(* Stoppen vom Prozess welches über den Automat ausgelöst wurde *)
	IF xTmpProcMachineStop THEN
		(* Step  function station stop  *)
		CASE iStepActionStop OF
		(* Überprüfe zuerst den Zustand des Prozesses ob es überhaupt zulässt, den Prozess zu stoppen *)
		1:	xTmp:=	TProcess.T_Ctrle.xRdy
					AND NOT(TProcess.T_Ctrle.xStop)
					AND NOT(TProcess.T_Ctrle.xDone)
					AND NOT(TProcess.T_Ctrle.xError)
					AND NOT(TProcess.T_Ctrle.xAbordProcess);
			IF xTmp THEN
				iStepActionStop:=10;
			(* not ready to execute stop *)
			ELSE iStepActionStop:=95; END_IF
		10:	TProcess.T_Ctrle.xStop:=TRUE;
			(* next step *)
			iStepActionStop:=20;
			xStepActionDoneStop:=FALSE;
		(* wait confirmation *)
		20:	T_ExchgParam.T_Visu.T_Message.iState:=232;	(* Warnung: Unverzüglicher Zyklus-Stopp ! *)
			IF NOT(xStepActionDoneStop) THEN
			(* release execution *)
				xStepActionDoneStop:=TRUE;
			ELSE
				IF NOT(TProcess.T_Ctrle.xStop) AND TProcess.T_Ctrle.xDone THEN
					(* Für Maschinenreferenzieren und Wstk Entlade Prozess wird der Prozess beendet *)
					xProcessAbordet:=TRUE;
					iStepActionStop:=90;
					xStepActionDoneStop:=FALSE;
					T_ExchgParam.T_Visu.T_Message.iState:=236;	(* Warnung: Prozess wurde gestoppt ! *)
				END_IF;
			END_IF;
		(* action done *)
		90:	xTmpProcMachineStop:=FALSE;
		(* function not ready *)
		95:	xTmpProcMachineStop:=FALSE;
		END_CASE;
	END_IF;
END_ACTION
ACTION VisuFunction_ProfileManagement:
(* Erstmalige Kopiervorgang der Profile *)
	IF xAction_CopyProfileToProcess THEN
		(* Set copy action *)
		CASE iStepAction OF
		(* Set default value *)
		1:	xFctSetDefaultValueStaticProfile(ptrT_DefaultProfileParameter:=ADR(T_Profile.T_DefaultProfileParameter));
			(* Init. display value *)
			xProfileFileNotFoundSt1:=FALSE;
			xWrongProfilNameReadedSt1:=FALSE;
			xProfileFileWrongSyntaxSt1:=FALSE;
			xProfileFileWrongSyntax:=FALSE;
			iStepAction:=2; (* Überprüfe zuerst als nächstes ob das USB Stick ansprechbar ist *)
		(* check first if USB-Stick exist *)
		2:	T_Profile.T_Ctrle.iFunction:=3;	(* check if the USB-Stick exist *)
			T_Profile.T_Ctrle.xExecute:=TRUE;
			iStepAction:=3;
		3:	IF NOT(T_Profile.T_Ctrle.xExecute) AND T_Profile.T_Ctrle.xDone THEN
				(* USB Stick exist *)
				iStepAction:=4;
			END_IF;
			IF NOT(T_Profile.T_Ctrle.xExecute) AND T_Profile.T_Ctrle.xErr THEN
				(* USB-Stick does not exist *)
				T_ExchgParam.T_Visu.T_Message.iState:=0;	(* Meldung zurücksetzen *)
				T_Profile.T_Ctrle.xReset:=TRUE;
				iStepAction:=98;
			END_IF;
		(* Read First all exist Profilname for manage the profile  *)
		4:	T_Profile.T_Ctrle.sPathAndFileName:='PROFILE\';
			T_Profile.T_Ctrle.iFunction:=6;
			T_Profile.T_Ctrle.xExecute:=TRUE;
			iStepAction:=5;
		5:	IF NOT(T_Profile.T_Ctrle.xExecute) AND T_Profile.T_Ctrle.xDone THEN
				(* all readed profile are ok *)
				iStepAction:=10;
			END_IF;
			IF NOT(T_Profile.T_Ctrle.xExecute) AND T_Profile.T_Ctrle.xErr THEN
				(* Wrong Syntax-->1 File of Profile is corrupted *)
				T_ExchgParam.T_Visu.T_Message.iState:=0;	(* Meldung zurücksetzen *)
				T_Profile.T_IDProfileStation[1].iNumber:=1;
				T_Profile.T_IDProfileStation[1].sName:='Default';
				T_Profile.T_Ctrle.xReset:=TRUE;
				xProfileFileWrongSyntax:=TRUE;
				iStepAction:=90;
			END_IF;
		(* activ reading profile file *)
		10:	IF T_NovRam.T_Parameter.T_StationWork[gciStationSt1].T_InfoProcess.iProfile > 0 AND T_NovRam.T_Parameter.T_StationWork[gciStationSt1].T_InfoProcess.iProfile <= csiMaxProfile THEN
				T_Profile.T_Ctrle.sPathAndFileName:='PROFILE\';
				T_Profile.T_Id.iNumber:=T_NovRam.T_Parameter.T_StationWork[gciStationSt1].T_InfoProcess.iProfile;
				T_Profile.T_Id.sName:=T_NovRam.T_Parameter.T_StationWork[gciStationSt1].T_InfoProcess.sProfileName;
				T_Profile.T_Ctrle.iFunction:=4;	(* read the profile file *)
				T_Profile.T_Ctrle.xExecute:=TRUE;
				(* next step *)
				iStepAction:=20;
			ELSE iStepAction:=25; END_IF
		20:	IF NOT T_Profile.T_Ctrle.xExecute AND T_Profile.T_Ctrle.xDone THEN
				(* Setzen des aktuellen Prozessabbild welches vom NovRAM ist *)
				T_Profile.T_LoadProfileParameter:=T_Profile.T_CopyProfileParameter;
				T_ExchgParam.T_StationCommon.T_Param_StationWork.T_InfoProcess.iProfile:=T_NovRam.T_Parameter.T_StationWork[gciStationSt1].T_InfoProcess.iProfile;
				T_ExchgParam.T_StationCommon.T_Param_StationWork.T_InfoProcess.sProfileName:=T_Profile.T_Id.sName;
				garPositionEndProcCalc[gciStationSt1]:=T_NovRam.T_Parameter.arZ1AxisCalcEndPosSaveProfile[gciStationSt1,T_NovRam.T_Parameter.T_StationWork[gciStationSt1].T_InfoProcess.iProfile];
				garCentringEndProcCalc[gciStationSt1]:=T_NovRam.T_Parameter.arZ1CentringCalcEndPosSaveProfile[gciStationSt1,T_NovRam.T_Parameter.T_StationWork[gciStationSt1].T_InfoProcess.iProfile];
				(* check if the read name of the profil file is the same as the save name *)
				IF (T_Profile.T_Ctrle.sProfileName <> T_Profile.T_Id.sName) THEN
					(* overwrite the profilname with the name wrote in the file *)
					T_NovRam.T_Parameter.T_StationWork[gciStationSt1].T_InfoProcess.sProfileName:=T_Profile.T_Ctrle.sProfileName;
					T_Profile.T_IDProfileStation[T_NovRam.T_Parameter.T_StationWork[gciStationSt1].T_InfoProcess.iProfile].sName:=T_Profile.T_Ctrle.sProfileName;
					xWrongProfilNameReadedSt1:=TRUE;
				END_IF;
				(* next step *)
				iStepAction:=90;
			END_IF
			IF T_Profile.T_Ctrle.xErr THEN
				iToLoadProfileNrSt1:=T_Profile.T_Id.iNumber;
				sToLoadProfileNameSt1:=T_Profile.T_Id.sName;
				IF (T_Profile.T_Ctrle.udiErrorID <> 16#F2000) THEN
					(* Profile file not founded *)
					xProfileFileNotFoundSt1:=TRUE;
				ELSE
					(* wrong syntax of readed Profile file *)
					xProfileFileWrongSyntaxSt1:=TRUE;
				END_IF;
				(* activ reset *)
				T_Profile.T_Ctrle.xReset:=TRUE;
				(* next step *)
				iStepAction:=25;
			END_IF
		(* waiting flag *)
		25:	IF NOT T_Profile.T_Ctrle.xReset AND T_Profile.T_Ctrle.xDone THEN
				IF (T_Profile.T_Id.iNumber = 1) THEN
					T_Profile.T_LoadProfileParameter:=T_Profile.T_DefaultProfileParameter;
					T_ExchgParam.T_StationCommon.T_Param_StationWork.T_InfoProcess.iProfile:=1;
					T_ExchgParam.T_StationCommon.T_Param_StationWork.T_InfoProcess.sProfileName:='Default';
					(* erase name *)
					T_Profile.T_IDProfileStation[1].sName:='Default';
					T_NovRam.T_Parameter.T_StationWork[gciStationSt1].T_InfoProcess.iProfile:=1;
					T_NovRam.T_Parameter.T_StationWork[gciStationSt1].T_InfoProcess.sProfileName:='Default';
					iStepAction:=90;
				ELSE
					(* erase name *)
					T_Profile.T_IDProfileStation[1].sName:='Default';
					T_NovRam.T_Parameter.T_StationWork[gciStationSt1].T_InfoProcess.iProfile:=1;
					T_NovRam.T_Parameter.T_StationWork[gciStationSt1].T_InfoProcess.sProfileName:='Default';
					iStepAction:=26;
				END_IF;
			END_IF
		(* activ reading profile file *)
		26:	T_Profile.T_Ctrle.sPathAndFileName:='PROFILE\';
			T_Profile.T_Id.iNumber:=1;
			T_Profile.T_Id.sName:='Default';
			T_Profile.T_Ctrle.iFunction:=4;	(* read the profile file *)
			T_Profile.T_Ctrle.xExecute:=TRUE;
			(* next step *)
			iStepAction:=20;
		(* End function *)
		90:	xTmp:=	xProfileFileNotFoundSt1 OR xWrongProfilNameReadedSt1 OR 	xProfileFileWrongSyntaxSt1 OR xProfileFileWrongSyntax;
			IF xTmp THEN
				IF xProfileFileNotFoundSt1 THEN
					T_ExchgParam.T_SafetyCtrl.diSetForceErrorNr:=(gciStationSt1 * 1000000) + 16#F301;	(* Datei für zu ladendes Profil nicht gefunden *)
				ELSE
					IF xWrongProfilNameReadedSt1 THEN
						T_ExchgParam.T_SafetyCtrl.diSetForceErrorNr:=(gciStationSt1 * 1000000) + 16#F303;	(* Profilname von Datei ist anders als geladenes Profil *)
					END_IF;
					IF xProfileFileWrongSyntaxSt1 THEN
						T_ExchgParam.T_SafetyCtrl.diSetForceErrorNr:=(gciStationSt1 * 1000000) + 16#F304;	(* Syntaxfehler von zu ladendes Profil *)
					END_IF;
					IF xProfileFileWrongSyntax THEN
						T_ExchgParam.T_SafetyCtrl.diSetForceErrorNr:=16#F303;	(* Syntaxfehler mindestens einer Profildatei beim lesen aller Profile *)
					END_IF;
				END_IF;
				T_ExchgParam.T_SafetyCtrl.xSetForceError:=TRUE;
				xProfileFileNotFoundSt1:=xWrongProfilNameReadedSt1:=xProfileFileWrongSyntaxSt1:=FALSE;
				xProfileFileWrongSyntax:=FALSE;
			END_IF;
			T_Visu.T_CtrleAction.xDone:=TRUE;
			T_Visu.T_CtrleAction.xErr:=FALSE;
			T_Visu.T_CtrleAction.udiErrorID:=16#0;
			xAction_CopyProfileToProcess:=FALSE;
			xUpdateProfileList:=TRUE;
		(* USB-Stick is missing  *)
		98:	T_Visu.T_CtrleAction.xDone:=TRUE;
			T_Visu.T_CtrleAction.xNotReady:=FALSE;
			T_Profile.T_Ctrle.xReset:=T_Profile.T_Ctrle.xErr;
			T_ExchgParam.T_SafetyCtrl.xSetForceError:=TRUE;
			T_ExchgParam.T_SafetyCtrl.diSetForceErrorNr:=16#F300;	(* USB-Stick konnte nicht gefunden werden für Profil lesen/schreiben *)
			T_Visu.T_CtrleAction.xErr:=FALSE;
			T_Visu.T_CtrleAction.udiErrorID:=0;
			xAction_CopyProfileToProcess:=FALSE;
		END_CASE
	END_IF

(* Laden eines ausgewählten Profil in den Prozessabbild *)
	IF xAction_LoadProfile THEN
		(* Step import/export profile value *)
		CASE iStepAction OF
		1:	IF NOT(T_NovRAM.T_Parameter.T_Machine.T_ParamSystem.xActive_ProfilLoadNormalMode) AND
			     NOT(gT_SafetyStatus.xSetupOperateModeActive) THEN
				T_ExchgParam.T_Visu.T_Message.iState:=250;	(* Warning: Laden Profile im Automat ist der Parameter gesperrt ! *)
				iStepAction:=90;
				RETURN;
			END_IF;
			T_ExchgParam.T_Visu.T_Message.iState:=104;	(* Aufforderung: Bestätigen Profil laden <Enter>, abbrechen <Esc> ? *)
			xWrongProfilNameReaded:=FALSE;
			xProfileFileNotFoundSt:=FALSE;
			xProfileFileWrongSyntax:=FALSE;
			(* next step *)
			iStepAction:=10;
		(* waiting for key <Enter> or <Esc> *)
		10:	IF RisingEdgeKeyPanel_Enter.Q THEN
				(* Display message transfering *)
				T_ExchgParam.T_Visu.T_Message.iState:=4;	(* Info: Übertragung von Werten... *)
				tTimeOutAction:=TimerAction.ET+T#10s;
				iStepAction:=11;
			ELSE
				IF RisingEdgeKeyPanel_Esc.Q THEN
					iStepAction:=90;
					T_ExchgParam.T_Visu.T_Message.iState:=202;	(* Warnung: Aktion abgebrochen ! *)
				END_IF
			END_IF
			(* An other message has been displayed *)
			IF (T_ExchgParam.T_Visu.T_Message.iState<>4) AND (T_ExchgParam.T_Visu.T_Message.iState<>104) AND (T_ExchgParam.T_Visu.T_Message.iState<>202) THEN iStepAction:=90; END_IF
		(* check first if USB-Stick exist *)
		11:	T_Profile.T_Ctrle.iFunction:=3;	(* check if the USB-Stick exist *)
			T_Profile.T_Ctrle.xExecute:=TRUE;
			iStepAction:=12;
		12:	IF NOT(T_Profile.T_Ctrle.xExecute) AND T_Profile.T_Ctrle.xDone THEN
				(* USB Stick exist *)
				IF (T_Profile.T_IDProfileStation[T_ExchgParam.T_ProfileCommon.T_Id.iNumber].sName = '') THEN
					T_ExchgParam.T_Visu.T_Message.iState:=218;		(* Warnung: Profil existiert nicht ! *)
					iStepAction:=90;
				ELSE
					iStepAction:=20;
				END_IF;
			END_IF;
			IF NOT(T_Profile.T_Ctrle.xExecute) AND T_Profile.T_Ctrle.xErr THEN
				(* USB-Stick does not exist *)
				T_ExchgParam.T_Visu.T_Message.iState:=0;	(* Meldung zurücksetzen *)
				T_Profile.T_Ctrle.xReset:=TRUE;
				iStepAction:=98;
			END_IF;
		(* Init. reading profile file *)
		20:	(* Save Old Slide Reference Position *)
			T_Profile.T_Ctrle.sPathAndFileName:='PROFILE\';
			T_Profile.T_Id.iNumber:=T_ExchgParam.T_ProfileCommon.T_Id.iNumber;
			T_Profile.T_Id.sName:=T_Profile.T_IDProfileStation[T_ExchgParam.T_ProfileCommon.T_Id.iNumber].sName;
			T_Profile.T_Ctrle.iFunction:=4;	(* read the profile file *)
			T_Profile.T_Ctrle.xExecute:=TRUE;
			(* Display info message *)
			T_ExchgParam.T_Visu.T_Message.iState:=4;	(* Info: Übertragung von Werten... *)
			(* next step *)
			iStepAction:=30;
		(* waiting confirmation signal *)
		30:	T_ExchgParam.T_Visu.T_Message.iState:=4;	(* Info: Übertragung von Werten... *)
			IF NOT T_Profile.T_Ctrle.xExecute AND T_Profile.T_Ctrle.xDone THEN
			(* Copy profile to online value *)
				T_NovRam.T_Parameter.T_StationWork[gciStationSt1].T_StProcess:=T_Profile.T_CopyProfileParameter.T_ProzessData;
				T_NovRam.T_Parameter.T_StationWork[gciStationSt1].T_OnlineChange:=T_Profile.T_CopyProfileParameter.T_ProfileOnlineChange;
				T_Profile.T_LoadProfileParameter:=T_Profile.T_CopyProfileParameter;
				IF (T_NovRam.T_Parameter.T_StationWork[gciStationSt1].T_InfoProcess.iProfile <> T_ExchgParam.T_ProfileCommon.T_Id.iNumber) THEN
					(* Anderes Profile geladen und deshalb muss der entsprechende Zählerstand des geladenen Profil übernommen werden *)
					garPositionEndProcCalc[gciStationSt1]:=T_NovRam.T_Parameter.arZ1AxisCalcEndPosSaveProfile[gciStationSt1,T_ExchgParam.T_ProfileCommon.T_Id.iNumber];
					garCentringEndProcCalc[gciStationSt1]:=T_NovRam.T_Parameter.arZ1CentringCalcEndPosSaveProfile[gciStationSt1,T_ExchgParam.T_ProfileCommon.T_Id.iNumber];
				END_IF;
				T_NovRam.T_Parameter.T_StationWork[gciStationSt1].T_InfoProcess.iProfile:=T_ExchgParam.T_ProfileCommon.T_Id.iNumber;
				T_NovRam.T_Parameter.T_StationWork[gciStationSt1].T_InfoProcess.sProfileName:=T_Profile.T_Id.sName;
				T_ExchgParam.T_ProfileCommon.T_OnlineChange.T_Data:=T_Profile.T_LoadProfileParameter.T_ProfileOnlineChange;
				T_ExchgParam.T_ProfileCommon.T_Id.sName:=T_Profile.T_Id.sName;
				T_ExchgParam.T_StationCommon.T_Param_StationWork.T_StProcess:=T_Profile.T_LoadProfileParameter.T_ProzessData;
				(* check if the read name of the profil file is the same as the save name *)
				IF (T_Profile.T_Ctrle.sProfileName <> T_Profile.T_Id.sName) THEN
					(* overwrite the profilname with the name wrote in the file *)
					T_NovRam.T_Parameter.T_StationWork[gciStationSt1].T_InfoProcess.sProfileName:=T_Profile.T_Ctrle.sProfileName;
					T_ExchgParam.T_ProfileCommon.T_Id.sName:=T_Profile.T_Ctrle.sProfileName;
					T_Profile.T_IDProfileStation[T_ExchgParam.T_ProfileCommon.T_Id.iNumber].sName:=T_Profile.T_Ctrle.sProfileName;
					xWrongProfilNameReaded:=TRUE;
				END_IF;
				(* next step *)
				iStepAction:=40;
			END_IF
			IF T_Profile.T_Ctrle.xErr THEN
				iToLoadProfileNrSt:=T_Profile.T_Id.iNumber;
				sToLoadProfileNameSt:=T_Profile.T_Id.sName;
				(* activ reset *)
				T_Profile.T_Ctrle.xReset:=TRUE;
				IF (T_Profile.T_Ctrle.udiErrorID <> 16#F2000) THEN
					(* Profile file not founded *)
					xProfileFileNotFoundSt:=TRUE;
					T_ExchgParam.T_ProfileCommon.T_Id.sName:='';
					(* Profile will be erased from the profile list *)
					T_Profile.T_IDProfileStation[T_ExchgParam.T_ProfileCommon.T_Id.iNumber].sName:='';
					xUpdateProfileList:=TRUE;
					(* next step *)
					iStepAction:=90;
				ELSE
					(* wrong syntax of readed Profile file *)
					xProfileFileWrongSyntax:=TRUE;
					(* next step *)
					iStepAction:=90;
				END_IF;
			END_IF
		(* save profile number *)
		40:	(* save profile number to process value *)
			T_ExchgParam.T_StationCommon.T_Param_StationWork.T_InfoProcess.iProfile:=T_ExchgParam.T_ProfileCommon.T_Id.iNumber;
			T_ExchgParam.T_StationCommon.T_Param_StationWork.T_InfoProcess.sProfileName:=T_ExchgParam.T_ProfileCommon.T_Id.sName;
			xUpdateHandlingConfig:=TRUE;
			(* activ next step *)
			iStepAction:=50;
		(* active saving data NovRAM *)
		50:	xAction_SaveNovRAM:=TRUE;
			xBlockSetNovRamAction_End:=TRUE;
			iStepActionNovRam:=1;
			(* next step *)
			iStepAction:=60;
		(* waiting confirm saving NovRAM action *)
		60:	IF NOT xAction_SaveNovRAM THEN
				T_ExchgParam.T_Visu.T_Message.iState:=54;	(* Info: Profil wurde geladen ! *)
				IF NOT(xProfileFileNotFoundSt) THEN
					iStepAction:=90;
				ELSE
					iStepAction:=90;
				END_IF;
			END_IF;
		(* save done *)
		90:	IF xProfileFileNotFoundSt OR xWrongProfilNameReaded OR xProfileFileWrongSyntax THEN
				IF xProfileFileNotFoundSt THEN
					T_ExchgParam.T_SafetyCtrl.diSetForceErrorNr:=(gciStationSt1 * 1000000) + 16#F301;	(* Datei für zu ladendes Profil nicht gefunden *)
				ELSE
					IF xWrongProfilNameReaded THEN
						T_ExchgParam.T_SafetyCtrl.diSetForceErrorNr:=(gciStationSt1 * 1000000) + 16#F303;	(* Profilname von Datei ist anders als geladenes Profil *)
					ELSE
						T_ExchgParam.T_SafetyCtrl.diSetForceErrorNr:=(gciStationSt1 * 1000000) + 16#F304;	(* Syntaxfehler von zu ladendes Profil *)
					END_IF;
				END_IF;
				T_ExchgParam.T_SafetyCtrl.xSetForceError:=TRUE;
				xProfileFileNotFoundSt:=xWrongProfilNameReaded:=xProfileFileWrongSyntax:=FALSE;
			END_IF;
			T_Visu.T_CtrleAction.xDone:=TRUE;
			T_Visu.T_CtrleAction.xNotReady:=FALSE;
			T_Visu.T_CtrleAction.xErr:=FALSE;
			T_Visu.T_CtrleAction.udiErrorID:=0;
			xAction_LoadProfile:=FALSE;
		(* USB-Stick is missing  *)
		98:	T_Visu.T_CtrleAction.xDone:=TRUE;
			T_Visu.T_CtrleAction.xNotReady:=FALSE;
			T_Profile.T_Ctrle.xReset:=T_Profile.T_Ctrle.xErr;
			T_ExchgParam.T_SafetyCtrl.xSetForceError:=TRUE;
			T_ExchgParam.T_SafetyCtrl.diSetForceErrorNr:=(gciStationSt1 * 1000000) + 16#F300;	(* USB-Stick konnte nicht gefunden werden für Profil lesen/schreiben *)
			T_Visu.T_CtrleAction.xErr:=FALSE;
			T_Visu.T_CtrleAction.udiErrorID:=0;
			xAction_LoadProfile:=FALSE;
		END_CASE
	ELSE
		IF NOT(xAction_CopyProfileToProcess) THEN
			IF (T_NovRam.T_Parameter.T_StationWork[1].T_InfoProcess.iProfile >= 1) AND (T_NovRam.T_Parameter.T_StationWork[1].T_InfoProcess.iProfile <= 100) THEN
				T_NovRam.T_Parameter.arZ1AxisCalcEndPosSaveProfile[gciStationSt1,T_NovRam.T_Parameter.T_StationWork[1].T_InfoProcess.iProfile]:=garPositionEndProcCalc[gciStationSt1];
				T_NovRam.T_Parameter.arZ1CentringCalcEndPosSaveProfile[gciStationSt1,T_NovRam.T_Parameter.T_StationWork[1].T_InfoProcess.iProfile]:=garCentringEndProcCalc[gciStationSt1];
			END_IF;
		END_IF;
	END_IF

(* Speichern eines ausgewählten Profils *)
	IF xAction_SaveProfile THEN
		(* Step saving NovRAM *)
		CASE iStepAction OF
		(* check first if USB-Stick exist *)
		1:	T_Profile.T_Ctrle.iFunction:=3;	(* check if the USB-Stick exist *)
			T_Profile.T_Ctrle.xExecute:=TRUE;
			iStepAction:=2;
		2:	IF NOT(T_Profile.T_Ctrle.xExecute) AND T_Profile.T_Ctrle.xDone THEN
				(* USB Stick exist *)
				iStepAction:=10;
			END_IF;
			IF NOT(T_Profile.T_Ctrle.xExecute) AND T_Profile.T_Ctrle.xErr THEN
				(* USB-Stick does not exist *)
				T_ExchgParam.T_Visu.T_Message.iState:=0;	(* Meldung zurücksetzen *)
				T_Profile.T_Ctrle.xReset:=TRUE;
				iStepAction:=98;
			END_IF;
		(* Display message to ask for confirmation *)
		10:	IF T_ExchgParam.T_ProfileCommon.T_Id.iNumber > 1 THEN
				IF T_ExchgParam.T_ProfileCommon.T_Id.sName <> '' THEN
					iTmp:=  iFctExistProfileName(	sProfileName:=T_ExchgParam.T_ProfileCommon.T_Id.sName,
												ptrProfileList:=ADR(T_Profile.T_IDProfileStation));
					IF iTmp = T_ExchgParam.T_ProfileCommon.T_Id.iNumber OR iTmp = 0 THEN
						IF (T_ExchgParam.T_StationCommon.T_Param_StationWork.T_InfoProcess.iProfile = T_ExchgParam.T_ProfileCommon.T_Id.iNumber) THEN
							(* Display message 'ask for rewriting' *)
							T_ExchgParam.T_Visu.T_Message.iState:=105;	(* Aufforderung: Das Profil wird überschrieben <Enter>, abbrechen <Esc> ? *)
							(* next step *)
							iStepAction:=20;
						ELSE
							(* Display message 'confirm saving' *)
							T_ExchgParam.T_Visu.T_Message.iState:=103;	(* Aufforderung: Speichern bestätigen <Enter>, abbrechen <Esc> ? *)
							(* next step *)
							iStepAction:=20;
						END_IF
					ELSE
						T_ExchgParam.T_Visu.T_Message.iState:=219;		(* Warnung: Profil existiert schon, Daten nicht gespeichert ! *)
						iStepAction:=90;
					END_IF;
				(* Display message, 'Profile name not correct' *)
				ELSE	T_ExchgParam.T_Visu.T_Message.iState:=220;		(* Warnung: Profilname nicht korrekt ! *)
						iStepAction:=90;
				END_IF
			ELSE
				T_ExchgParam.T_Visu.T_Message.iState:=221;	(* Warnung: Default-Profilwerte können nicht geändert werden ! *)
				iStepAction:=90;
			END_IF
		(* waiting for confirmation key <Enter> or <Esc> *)
		20:	IF RisingEdgeKeyPanel_Enter.Q THEN
			(* Display message *)
				T_ExchgParam.T_Visu.T_Message.iState:=3;		(* Info: Start speichern... *)
				tTimeOutAction:=TimerAction.ET+T#10s;
				(* next step *)
				iStepAction:=30;
			ELSE
				IF RisingEdgeKeyPanel_Esc.Q THEN
					iStepAction:=90;
					T_ExchgParam.T_Visu.T_Message.iState:=202;	(* Warnung: Aktion abgebrochen ! *)
				END_IF
			END_IF
			(* An other message has been displayed *)
			IF (T_ExchgParam.T_Visu.T_Message.iState<>3) AND (T_ExchgParam.T_Visu.T_Message.iState<>103) AND
			     (T_ExchgParam.T_Visu.T_Message.iState<>105) AND (T_ExchgParam.T_Visu.T_Message.iState<>202) THEN iStepAction:=90; END_IF
		30:	(* activ saving profile file *)
			T_Profile.T_Ctrle.sPathAndFileName:='PROFILE\';
			T_Profile.T_Id.iNumber:=T_ExchgParam.T_ProfileCommon.T_Id.iNumber;
			T_Profile.T_Id.sName:=T_ExchgParam.T_ProfileCommon.T_Id.sName;
			T_Profile.T_Ctrle.iFunction:=5;	(* write the profile file *)
			T_Profile.T_Ctrle.xExecute:=TRUE;
			T_Profile.T_CopyProfileParameter.T_ProzessData:=T_NovRam.T_Parameter.T_StationWork[gciStationSt1].T_StProcess;
			T_Profile.T_CopyProfileParameter.T_ProfileOnlineChange:=T_NovRam.T_Parameter.T_StationWork[gciStationSt1].T_OnlineChange;
			(* next step *)
			iStepAction:=40;
		(* waiting signal and start saving data in NovRAM *)
		40:	T_ExchgParam.T_Visu.T_Message.iState:=3;		(* Info: Start speichern... *)
			IF NOT(T_Profile.T_Ctrle.xExecute) AND T_Profile.T_Ctrle.xDone THEN
				T_Profile.T_IDProfileStation[T_ExchgParam.T_ProfileCommon.T_Id.iNumber]:=T_ExchgParam.T_ProfileCommon.T_Id;
				(* Process profile value = file profile value *)
				IF (T_ExchgParam.T_ProfileCommon.T_Id.iNumber = T_NovRam.T_Parameter.T_StationWork[gciStationSt1].T_InfoProcess.iProfile) THEN
					(* Beim speichern eines Profils darf dies nicht durchgeführt werden, sofern nicht das gleiche Profil gespeichert wird wo schon geladen ist,
					    weil sonst der Blaue Profilebalken überschrieben wird *)
					T_ExchgParam.T_StationCommon.T_Param_StationWork.T_InfoProcess.sProfileName:=T_ExchgParam.T_ProfileCommon.T_Id.sName;
					T_Profile.T_LoadProfileParameter:=T_Profile.T_ProcProfileParameter;
					T_NovRam.T_Parameter.T_StationWork[gciStationSt1].T_InfoProcess.sProfileName:=T_ExchgParam.T_ProfileCommon.T_Id.sName;
				END_IF
				(* page profile, update profile list *)
				xUpdateProfileList:=TRUE;
				(* next step *)
				iStepAction:=50;
			END_IF
			IF T_Profile.T_Ctrle.xErr THEN
				iStepAction:=98;
			END_IF
		(* save Image in NovRAM *)
		50:	T_NovRAM.T_Ctrle.xExecute:=TRUE;
			T_NovRAM.T_Ctrle.iFunction:=2;
			(* next Step *)
			iStepAction :=60;
			xStepActionDone:=FALSE;
		(* wait save confirmation *)
		60:	IF NOT(xStepActionDone) THEN
				T_NovRAM.T_Ctrle.xExecute:=FALSE;
				(* confirm Step *)
				xStepActionDone:=TRUE;
			ELSE
				IF T_NovRAM.T_Ctrle.xDone THEN
				(* next Step *)
					iStepAction :=90;
					xStepActionDone:=FALSE;
					T_ExchgParam.T_Visu.T_Message.iState:=55;	(* Info: Profil wurde gespeichert ! *)
				ELSE	IF T_NovRAM.T_Ctrle.xErr THEN
							iStepAction:=99;
							xStepActionDone:=FALSE;
						END_IF
				END_IF
			END_IF
		(* save done *)
		90:	T_Visu.T_CtrleAction.xDone:=TRUE;
			T_Visu.T_CtrleAction.xNotReady:=FALSE;
			T_Visu.T_CtrleAction.xErr:=FALSE;
			T_Visu.T_CtrleAction.udiErrorID:=0;
			xAction_SaveProfile:=FALSE;
		(* NovRAM not ready *)
		95:	TimerNotReady(IN:=TRUE);
			xAction_SaveProfile:=FALSE;
		(* USB-Stick is missing or directory is missing *)
		98:	T_Visu.T_CtrleAction.xDone:=TRUE;
			T_Visu.T_CtrleAction.xNotReady:=FALSE;
			T_Profile.T_Ctrle.xReset:=T_Profile.T_Ctrle.xErr;
			IF T_Profile.T_Ctrle.xErr THEN
				T_ExchgParam.T_SafetyCtrl.diSetForceErrorNr:=(gciStationSt1 * 1000000) + 16#F306;	(* Profil konnte nicht gespeichert werden da Verzeichnis fehlt *)
			ELSE
				T_ExchgParam.T_SafetyCtrl.diSetForceErrorNr:=(gciStationSt1 * 1000000) + 16#F300;	(* USB-Stick konnte nicht gefunden werden für Profil lesen/schreiben *)
			END_IF;
			T_ExchgParam.T_SafetyCtrl.xSetForceError:=TRUE;
			T_Visu.T_CtrleAction.xErr:=FALSE;
			T_Visu.T_CtrleAction.udiErrorID:=0;
			xAction_SaveProfile:=FALSE;
		(* error *)
		99:	T_Visu.T_CtrleAction.xDone:=TRUE;
			T_Visu.T_CtrleAction.xNotReady:=FALSE;
			T_Visu.T_CtrleAction.xErr:=FALSE;
			T_Visu.T_CtrleAction.udiErrorID:=0;
			xAction_SaveProfile:=FALSE;
			IF T_HDD.T_Ctrle.xErr THEN T_HDD.T_Ctrle.xReset:=TRUE; END_IF
			IF T_Profile.T_Ctrle.xErr THEN T_Profile.T_Ctrle.xReset:=TRUE; END_IF
			IF T_NovRAM.T_Ctrle.xErr THEN T_NovRAM.T_Ctrle.xReset:=TRUE; END_IF;
			T_ExchgParam.T_SafetyCtrl.diSetForceErrorNr:=(gciStationSt1 * 1000000) + 16#F305;	(* NovRAM Speicher Fehlerhaft *)
			T_ExchgParam.T_SafetyCtrl.xSetForceError:=TRUE;
		END_CASE
	END_IF

(* Löschen eines ausgewählten Profil *)
	IF xActionDeleteProfile THEN
		(* Step delete profile *)
		CASE iStepAction OF
		(* Profile number could not be 1 *)
		1:	IF T_ExchgParam.T_ProfileCommon.T_Id.iNumber < 2 THEN
				T_ExchgParam.T_Visu.T_Message.iState:=222;	(* Warnung: Default Profil kann nicht gelöscht werden ! *)
				iStepAction:=90;
			ELSIF T_ExchgParam.T_StationCommon.T_Param_StationWork.T_InfoProcess.iProfile = T_ExchgParam.T_ProfileCommon.T_Id.iNumber THEN
				T_ExchgParam.T_Visu.T_Message.iState:=223;	(* Warnung: Geladenes Profil kann nicht gelöscht werden ! *)
				iStepAction:=90;
			ELSE
				iStepAction:=2;
			END_IF;
		(* check first if USB-Stick exist *)
		2:	T_Profile.T_Ctrle.iFunction:=3;	(* check if the USB-Stick exist *)
			T_Profile.T_Ctrle.xExecute:=TRUE;
			iStepAction:=3;
		3:	IF NOT(T_Profile.T_Ctrle.xExecute) AND T_Profile.T_Ctrle.xDone THEN
				(* USB Stick exist *)
				iStepAction:=20;
			END_IF;
			IF NOT(T_Profile.T_Ctrle.xExecute) AND T_Profile.T_Ctrle.xErr THEN
				(* USB-Stick does not exist *)
				T_ExchgParam.T_Visu.T_Message.iState:=0;	(* Meldung löschen *)
				T_Profile.T_Ctrle.xReset:=TRUE;
				iStepAction:=98;
			END_IF;
		(* no code, waiting timeout *)
		10:	IF TimerAction.Q THEN xActionDeleteProfile:=FALSE; END_IF;
		20:	T_ExchgParam.T_Visu.T_Message.iState:=106;	(* Aufforderung: Bestätigen Profil löschen <Enter>, abbrechen <Esc> ? *)
			(* next step *)
			iStepAction:=30;
		(* waiting for key <Enter> or <Esc> *)
		30:	IF RisingEdgeKeyPanel_Enter.Q THEN
				T_ExchgParam.T_Visu.T_Message.iState:=5;	(* Info: Start löschen... *)
				(* next step *)
				iStepAction:=40;
			ELSE
				IF RisingEdgeKeyPanel_Esc.Q THEN
					iStepAction:=90;
					T_ExchgParam.T_Visu.T_Message.iState:=202;	(* Warnung: Aktion abgebrochen ! *)
				END_IF
			END_IF
			(* An other message has been displayed *)
			IF (T_ExchgParam.T_Visu.T_Message.iState<>5) AND (T_ExchgParam.T_Visu.T_Message.iState<>106) AND (T_ExchgParam.T_Visu.T_Message.iState<>202) THEN iStepAction:=90; END_IF
		(* Init. deleting profile file *)
		40:	T_Profile.T_Ctrle.sPathAndFileName:='PROFILE\';
			T_Profile.T_Id.iNumber:=T_ExchgParam.T_ProfileCommon.T_Id.iNumber;
			T_Profile.T_Ctrle.iFunction:=8;	(* delete the profile file *)
			T_Profile.T_Ctrle.xExecute:=TRUE;
			iStepAction:=50;
		50:	IF NOT(T_Profile.T_Ctrle.xExecute) AND T_Profile.T_Ctrle.xDone OR T_Profile.T_Ctrle.xErr THEN
				T_Profile.T_Ctrle.xReset:=T_Profile.T_Ctrle.xErr;
				(* Profile will be erased from the profile list *)
				T_Profile.T_IDProfileStation[T_ExchgParam.T_ProfileCommon.T_Id.iNumber].sName:='';
				xUpdateProfileList:=TRUE;
				IF T_Profile.T_Ctrle.xErr THEN
					T_ExchgParam.T_Visu.T_Message.iState:=224;	(* Warnung: Zu löschendes Profil existiert nicht ! *)
					(* next step *)
					iStepAction:=90;
					xStepActionDone:=FALSE;
				ELSE
					(* next step *)
					iStepAction:=70;
					xStepActionDone:=FALSE;
					T_ExchgParam.T_Visu.T_Message.iState:=56;	(* Info: Profil wurde gelöscht ! *)
				END_IF;
			END_IF
		(* active saving data NovRAM *)
		70:	(* Wenn ein Profil gelöscht wird, dann wird der Name auch in der Auswahl des Profilsnamen gelöscht *)
			T_ExchgParam.T_ProfileCommon.T_Id.sName:='';
			xAction_SaveNovRAM:=TRUE;
			xBlockSetNovRamAction_End:=TRUE;
			iStepActionNovRam:=1;
			(* next step *)
			iStepAction:=80;
		(* waiting confirm saving NovRAM action *)
		80:	IF NOT xAction_SaveNovRAM THEN iStepAction:=90; END_IF
		(* save done *)
		90:	T_Visu.T_CtrleAction.xDone:=TRUE;
			T_Visu.T_CtrleAction.xNotReady:=FALSE;
			T_Visu.T_CtrleAction.xErr:=FALSE;
			T_Visu.T_CtrleAction.udiErrorID:=0;
			xActionDeleteProfile:=FALSE;
		(* USB-Stick is missing  *)
		98:	T_Visu.T_CtrleAction.xDone:=TRUE;
			T_Visu.T_CtrleAction.xNotReady:=FALSE;
			T_Profile.T_Ctrle.xReset:=T_Profile.T_Ctrle.xErr;
			T_ExchgParam.T_SafetyCtrl.xSetForceError:=TRUE;
			T_ExchgParam.T_SafetyCtrl.diSetForceErrorNr:=(gciStationSt1 * 1000000) + 16#F302;	(* USB-Stick konnte nicht gefunden werden für Profil löschen *)
			T_Visu.T_CtrleAction.xErr:=FALSE;
			T_Visu.T_CtrleAction.udiErrorID:=0;
			xActionDeleteProfile:=FALSE;
		END_CASE;
	END_IF;
END_ACTION
ACTION VisuFunction_SafetyDoor:
(* Toggeln Maschinen- oder Lade- Tür Zuhaltung *)
	IF xMachineDoorUpGuardControlTogOnOff THEN
		(* set new page *)
		CASE iStepAction OF
		(* check ctrle visu *)
		1: 	(* activ next step *)
			iStepAction:=10;
			xStepActionDone:=FALSE;
		(* Set new page *)
		10:	IF xMachineDoorUpGuardControlTogOnOff THEN
				QxCabinDoorLock:=NOT(QxCabinDoorLock);
			END_IF;
			iStepAction:=90;
		(* override done *)
		90:	T_Visu.T_CtrleAction.xDone:=TRUE;
			T_Visu.T_CtrleAction.xNotReady:=FALSE;
			T_Visu.T_CtrleAction.xErr:=FALSE;
			T_Visu.T_CtrleAction.udiErrorID:=0;
			xMachineDoorUpGuardControlTogOnOff:=FALSE;
		END_CASE
	END_IF

(* Zustandausgabe von Maschinen und Ladetüre für die Visualisierung *)
	IF (T_Visu.T_PlcParam.dwActualPage = gT_PageNumber.iAutoMode_SafetyCheck) THEN
		(* Zustand 1 für Türe oben geschlossen: Obere Türe ist geschlossen *)
		xSecurityDoorUpCloseState:=	T_TwinSafeIn.IxCabinDoorCloseCh1 AND T_TwinSafeIn.IxCabinDoorCloseCh2 AND T_TwinSafeIn.IxCabinDoorClose AND
									NOT(T_TwinSafeIn.IxCabinDoorOpen);
		(* Zustand für Türe oben geöffnet: Obere Türe ist geöffnet und untere Türe kann geöffnet oder geschlossen sein *)
		xSecurityDoorUpOpenState:=	NOT(T_TwinSafeIn.IxCabinDoorCloseCh1) AND NOT(T_TwinSafeIn.IxCabinDoorCloseCh2) AND NOT(T_TwinSafeIn.IxCabinDoorClose) AND
									T_TwinSafeIn.IxCabinDoorOpen;
		IF xSecurityDoorUpCloseState THEN
			T_ExchgParam.T_SafetyCtrl.bMachineDoorUpState:=2;	(* MaschinenTüre oben geschlossen *)
		ELSIF xSecurityDoorUpOpenState THEN
			T_ExchgParam.T_SafetyCtrl.bMachineDoorUpState:=1;	(* MaschinenTüre oben geöffnet *)
		ELSE
			T_ExchgParam.T_SafetyCtrl.bMachineDoorUpState:=3;	(* MaschinenTüre oben Fehlverhalten *)
		END_IF;
		IF T_TwinSafeIn.IxCabinDoorCloseCh1 THEN
			T_ExchgParam.T_SafetyCtrl.bMachineDoorChannel1State:=2;	(* ON *)
		ELSE
			T_ExchgParam.T_SafetyCtrl.bMachineDoorChannel1State:=1;	(* OFF *)
		END_IF;
		IF T_TwinSafeIn.IxCabinDoorCloseCh2 THEN
			T_ExchgParam.T_SafetyCtrl.bMachineDoorChannel2State:=2;	(* ON *)
		ELSE
			T_ExchgParam.T_SafetyCtrl.bMachineDoorChannel2State:=1;	(* OFF *)
		END_IF;
		IF T_TwinSafeIn.IxCabinDoorOpen THEN
			T_ExchgParam.T_SafetyCtrl.bMachineDoorUpOpenState:=2;	(* ON *)
		ELSE
			T_ExchgParam.T_SafetyCtrl.bMachineDoorUpOpenState:=1;	(* OFF *)
		END_IF;
		IF T_TwinSafeIn.IxCabinDoorClose THEN
			T_ExchgParam.T_SafetyCtrl.bMachineDoorInductiveSensorState:=2;	(* ON *)
		ELSE
			T_ExchgParam.T_SafetyCtrl.bMachineDoorInductiveSensorState:=1;	(* OFF *)
		END_IF;
		IF QxCabinDoorLock AND NOT(IxCabinDoorLocked) THEN
			T_ExchgParam.T_SafetyCtrl.bMachineDoorGuardControlState:=2;		(* ON *)
		ELSIF NOT(QxCabinDoorLock) AND IxCabinDoorLocked THEN
			T_ExchgParam.T_SafetyCtrl.bMachineDoorGuardControlState:=1;		(* OFF *)
		ELSE
			T_ExchgParam.T_SafetyCtrl.bMachineDoorGuardControlState:=3;		(* Fehlverhalten *)
		END_IF;
	END_IF;
END_ACTION
ACTION VisuFunction_SetNewPage:
(* Set New page *)
	IF xSetNewPage THEN
		(* set new page *)
		CASE iStepAction OF
		(* check ctrle visu *)
		1: 	(* activ next step *)
			iStepAction:=10;
			xStepActionDone:=FALSE;
			xTmp:=	NOT(T_Visu.T_CtrleVisu.xDone)
					OR T_Visu.T_CtrleVisu.xExecute
					OR T_Visu.T_CtrleVisu.xErr;
			IF xTmp THEN iStepAction:=95; END_IF
		(* Set new page *)
		10:	T_Visu.T_CtrleVisu.iFunction:=1;
			T_Visu.T_CtrleVisu.xExecute:=TRUE;
			(* activ step *)
			iStepAction:=20;
			xStepActionDone:=FALSE;
		(* wait for changing page *)
		20:	IF NOT(xStepActionDone) THEN
			(* release execution *)
				T_Visu.T_CtrleVisu.xExecute:=FALSE;
				(* confirm step done *)
				xStepActionDone:=TRUE;
			ELSE
				IF T_Visu.T_CtrleVisu.xDone THEN
				(* activ next step *)
					iStepAction:=90;
					xStepActionDone:=FALSE;
				END_IF
				IF T_Visu.T_CtrleVisu.xErr THEN
				(* activ next error *)
					iStepAction:=99;
					xStepActionDone:=FALSE;
				END_IF
			END_IF
		(* override done *)
		90:	xBlockConfirmMessage:=TRUE;
			T_Visu.T_CtrleAction.xDone:=TRUE;
			T_Visu.T_CtrleAction.xNotReady:=FALSE;
			T_Visu.T_CtrleAction.xErr:=FALSE;
			T_Visu.T_CtrleAction.udiErrorID:=0;
			xSetNewPage:=FALSE;
		(* not ready *)
		95:	TimerNotReady(IN:=TRUE);
			xSetNewPage:=FALSE;
		(* error *)
		99:	T_Visu.T_CtrleAction.xDone:=FALSE;
			T_Visu.T_CtrleAction.xNotReady:=FALSE;
			T_Visu.T_CtrleAction.xErr:=TRUE;
			T_Visu.T_CtrleAction.udiErrorID:=16#F0000 + T_Visu.T_CtrleAction.iFunction;
			xSetNewPage:=FALSE;
		END_CASE
	END_IF
END_ACTION
ACTION VisuFunction_SetNewPageVertical:
(* Action Set main page auto/station + next/previous page vertical*)
	IF xNextPageVertical OR  xPreviousPageVertical THEN
		(* set next or previous page vertical *)
		CASE iStepAction OF
		(* check if page exist *)
		1:	(* init. variable *)
			iStepAction:=90;
			IF T_StartUp.T_State.xBlockChangeMovementVisu THEN RETURN; END_IF;
			(* vertical page navigation *)
			IF (T_Visu.T_PlcParam.dwActualPage > 1) AND (T_Visu.T_PlcParam.dwActualPage < 999) THEN
			(* array ranch 1 to 999 *)
				(* activ next page vertical *)
				IF xNextPageVertical THEN
					(* start page vertical *)
					iStepAction:=30;
					IF (T_Visu.T_PageIndex[T_Visu.T_PlcParam.dwActualPage+1].iIndexConfigPage) <> 0 THEN iStepAction:=10; END_IF
				END_IF
				(* activ previous page vertical *)
				IF xPreviousPageVertical THEN
					IF ((T_Visu.T_PageIndex[T_Visu.T_PlcParam.dwActualPage-1].iIndexConfigPage) <> 0) THEN
						iStepAction:=20;
					ELSE
						(* Set Last Page from Task *)
						iStepAction:=40;
					END_IF;
				END_IF
			END_IF
		(* next page vertical *)
		10:	(* activ step *)
			iStepAction:=80;
			xStepActionDone:=FALSE;
			T_Visu.T_PlcParam.dwSetNewPage:=T_Visu.T_PlcParam.dwActualPage+1;
			T_Visu.T_CtrleVisu.iFunction:=1;
			T_Visu.T_CtrleVisu.xExecute:=TRUE;
		(* previous page vertical *)
		20:	T_Visu.T_PlcParam.dwSetNewPage:=T_Visu.T_PlcParam.dwActualPage-1;
			T_Visu.T_CtrleVisu.iFunction:=1;
			T_Visu.T_CtrleVisu.xExecute:=TRUE;
			(* activ step *)
			iStepAction:=80;
			xStepActionDone:=FALSE;
		(* start page vertical *)
		30:	iTmp:=DWORD_TO_INT(T_Visu.T_PlcParam.dwActualPage);
			WHILE (iTmp MOD 10) <> 0 DO
				iTmp:=iTmp-1;
			END_WHILE
			T_Visu.T_PlcParam.dwSetNewPage:=iTmp;
			T_Visu.T_CtrleVisu.iFunction:=1;
			T_Visu.T_CtrleVisu.xExecute:=TRUE;
			(* activ step *)
			iStepAction:=80;
			xStepActionDone:=FALSE;
		40:	FOR ii:=1 TO 9 DO
				IF (T_Visu.T_PageIndex[T_Visu.T_PlcParam.dwActualPage+ii].iIndexConfigPage = 0) THEN
					T_Visu.T_PlcParam.dwSetNewPage:=T_Visu.T_PlcParam.dwActualPage+ii - 1;
					T_Visu.T_CtrleVisu.iFunction:=1;
					T_Visu.T_CtrleVisu.xExecute:=TRUE;
					(* activ step *)
					iStepAction:=80;
					xStepActionDone:=FALSE;
					EXIT;
				END_IF;
			END_FOR;
		(* wait for changing page *)
		80:	IF NOT(xStepActionDone) THEN
			(* release execution *)
				T_Visu.T_CtrleVisu.xExecute:=FALSE;
				(* confirm step done *)
				xStepActionDone:=TRUE;
			ELSE
				IF T_Visu.T_CtrleVisu.xDone THEN
				(* activ next step *)
					iStepAction:=90;
					xStepActionDone:=FALSE;
				END_IF
				IF T_Visu.T_CtrleVisu.xErr THEN
				(* activ next error *)
					iStepAction:=99;
					xStepActionDone:=FALSE;
				END_IF
			END_IF
		(* override done *)
		90:	xBlockConfirmMessage:=TRUE;
			T_Visu.T_CtrleAction.xDone:=TRUE;
			T_Visu.T_CtrleAction.xNotReady:=FALSE;
			T_Visu.T_CtrleAction.xErr:=FALSE;
			T_Visu.T_CtrleAction.udiErrorID:=0;
			xNextPageVertical:=FALSE;
			xPreviousPageVertical:=FALSE;
		(* not ready *)
		95:	TimerNotReady(IN:=TRUE);
			xNextPageVertical:=FALSE;
			xPreviousPageVertical:=FALSE;
		(* error *)
		99:	T_Visu.T_CtrleAction.xDone:=FALSE;
			T_Visu.T_CtrleAction.xNotReady:=FALSE;
			T_Visu.T_CtrleAction.xErr:=TRUE;
			T_Visu.T_CtrleAction.udiErrorID:=16#F0000 + T_Visu.T_CtrleAction.iFunction;
			xNextPageVertical:=FALSE;
			xPreviousPageVertical:=FALSE;
		END_CASE
	END_IF
END_ACTION
ACTION VisuFunction_SetParameterPage:
(* Set parameter page *)
	IF xSetParameterPage THEN
		(* set new page *)
		CASE iStepAction OF
		(* check ctrle visu *)
		1: 	(* activ next step *)
			iStepAction:=10;
			xStepActionDone:=FALSE;
			xTmp:=	NOT(T_Visu.T_CtrleVisu.xDone)
					OR T_Visu.T_CtrleVisu.xExecute
					OR T_Visu.T_CtrleVisu.xErr;
			IF xTmp THEN iStepAction:=95; END_IF
		(* Set new page *)
		10:	xUpdateStationParameter:=TRUE;
			T_Visu.T_CtrleVisu.iFunction:=1;
			T_Visu.T_CtrleVisu.xExecute:=TRUE;
			awSaveStateTaskBar[T_ExchgParam.T_Visu.bActiveSetupMode]:=T_ExchgParam.T_TouchScreenNavPanel.wState;
			(* activ step *)
			iStepAction:=20;
			xStepActionDone:=FALSE;
		(* wait for changing page *)
		20:	IF NOT(xStepActionDone) THEN
			(* release execution *)
				T_Visu.T_CtrleVisu.xExecute:=FALSE;
				(* confirm step done *)
				xStepActionDone:=TRUE;
			ELSE
				IF T_Visu.T_CtrleVisu.xDone THEN
				(* activ next step *)
					iStepAction:=90;
					xStepActionDone:=FALSE;
				END_IF
				IF T_Visu.T_CtrleVisu.xErr THEN
				(* activ next error *)
					iStepAction:=99;
					xStepActionDone:=FALSE;
				END_IF
			END_IF
		(* override done *)
		90:	xBlockConfirmMessage:=TRUE;
			T_Visu.T_CtrleAction.xDone:=TRUE;
			T_Visu.T_CtrleAction.xNotReady:=FALSE;
			T_Visu.T_CtrleAction.xErr:=FALSE;
			T_Visu.T_CtrleAction.udiErrorID:=0;
			xSetParameterPage:=FALSE;
		(* not ready *)
		95:	TimerNotReady(IN:=TRUE);
			xSetParameterPage:=FALSE;
		(* error *)
		99:	T_Visu.T_CtrleAction.xDone:=FALSE;
			T_Visu.T_CtrleAction.xNotReady:=FALSE;
			T_Visu.T_CtrleAction.xErr:=TRUE;
			T_Visu.T_CtrleAction.udiErrorID:=16#F0000 + T_Visu.T_CtrleAction.iFunction;
			xSetParameterPage:=FALSE;
		END_CASE
	END_IF
END_ACTION
ACTION VisuFunction_SetPreviousPage:
(* Set previous page *)
	IF xSetPreviousPage THEN
		(* set previous page *)
		CASE iStepAction OF
		(* check ctrle visu *)
		1: 	(* activ next step *)
			iStepAction:=10;
			xStepActionDone:=FALSE;
			xTmp:=	NOT(T_Visu.T_CtrleVisu.xDone)
					OR T_Visu.T_CtrleVisu.xExecute
					OR T_Visu.T_CtrleVisu.xErr;
			IF xTmp THEN iStepAction:=95; END_IF
		(* Set new page *)
		10:	xUpdateStationParameter:=TRUE;
			T_Visu.T_CtrleVisu.iFunction:=1;
			T_Visu.T_PlcParam.dwSetNewPage:=dwSaveActualPageTask[T_ExchgParam.T_Visu.bActiveSetupMode,iFct_GetBitNumber(wInputButton:=awSaveStateTaskBar[T_ExchgParam.T_Visu.bActiveSetupMode])];
			T_Visu.T_CtrleVisu.xExecute:=TRUE;
			(* activ step *)
			iStepAction:=20;
			xStepActionDone:=FALSE;
		(* wait for changing page *)
		20:	IF NOT(xStepActionDone) THEN
			(* release execution *)
				T_Visu.T_CtrleVisu.xExecute:=FALSE;
				(* confirm step done *)
				xStepActionDone:=TRUE;
			ELSE
				IF T_Visu.T_CtrleVisu.xDone THEN
				(* activ next step *)
					iStepAction:=90;
					xStepActionDone:=FALSE;
				END_IF
				IF T_Visu.T_CtrleVisu.xErr THEN
				(* activ next error *)
					iStepAction:=99;
					xStepActionDone:=FALSE;
				END_IF
			END_IF
		(* override done *)
		90:	xBlockConfirmMessage:=TRUE;
			T_Visu.T_CtrleAction.xDone:=TRUE;
			T_Visu.T_CtrleAction.xNotReady:=FALSE;
			T_Visu.T_CtrleAction.xErr:=FALSE;
			T_Visu.T_CtrleAction.udiErrorID:=0;
			xSetPreviousPage:=FALSE;
		(* not ready *)
		95:	TimerNotReady(IN:=TRUE);
			xSetPreviousPage:=FALSE;
		(* error *)
		99:	T_Visu.T_CtrleAction.xDone:=FALSE;
			T_Visu.T_CtrleAction.xNotReady:=FALSE;
			T_Visu.T_CtrleAction.xErr:=TRUE;
			T_Visu.T_CtrleAction.udiErrorID:=16#F0000 + T_Visu.T_CtrleAction.iFunction;
			xSetPreviousPage:=FALSE;
		END_CASE
	END_IF
END_ACTION
ACTION VisuFunction_Setup_Z_Axis:
(* Ausführen von Stationsfunktionen für das Einrichten der Z Achse für die Ersteinrichtung *)
	IF xStationSetupAxisZFunction THEN
		(* Step  function station  *)
		CASE iStepAction OF
		(* Überprüfe zuerst ob die Stationen bereit stehen  *)
		1:	(* For start the procedure, it need the system level *)
			IF (T_ExchgParam.T_Visu.T_Level.iActLevel <> 2) THEN
				T_ExchgParam.T_Visu.T_Message.iState:=216;	(* Warnung: Diese Parameter können nur auf SystemLevel geändert werden ! *)
				iStepAction:=90;
				RETURN;
			END_IF;
			xTmp:=	ptrActivStation^.TControl.xDone
					AND ptrActivStation^.TControl.xRdy
					AND NOT(ptrActivStation^.TControl.xExecute)
					AND NOT(ptrActivStation^.TControl.xError)
					AND NOT(ptrActivStation^.TControl.xStop);
			(* next step *)
			IF xTmp THEN
				T_ExchgParam.T_StationCommon.iZAxisFirstSetup_StepNr:=2;				(* Untere Anweisung durchführen!! *)
				T_ExchgParam.T_StationCommon.iZAxisFirstSetupStartButton_StepNr:=2;	(* Nachträglich Bitte StartTaste drücken! *)
				T_ExchgParam.T_StationCommon.iZAxisFirstSetup_ShowObjectNr:=2;
				iStepAction:=10;
				T_ExchgParam.T_Visu.T_Message.iState:=58;	(* Info: Funktion gestartet ! *)
			ELSE iStepAction:=95; END_IF
		(* Visu Ressource muss frei gegeben werden, da in dieser Prozedur noch zusätzliche VisuFunktionen benötigt werden *)
		10:	xTmpStationSetupAxisZFunction:=TRUE;
			iStepHelpVisuFunction:=1;
			T_StartUp.T_State.xBlockChangeMovementVisu:=TRUE;	(* Blockiere die Visu Navigation *)
			iStepAction:=90;
		(* action done *)
		90:	T_Visu.T_CtrleAction.xDone:=TRUE;
			T_Visu.T_CtrleAction.xNotReady:=FALSE;
			T_Visu.T_CtrleAction.xErr:=FALSE;
			T_Visu.T_CtrleAction.udiErrorID:=0;
			xStationSetupAxisZFunction:=FALSE;
		(* function not ready *)
		95:	TimerNotReady(IN:=TRUE);
			xStationSetupAxisZFunction:=FALSE;
		END_CASE
	ELSE
		IF NOT(xTmpStationSetupAxisZFunction) THEN
			T_ExchgParam.T_StationCommon.iZAxisFirstSetup_StepNr:=1;				(* Setzen der Z Nullstellung und ausmessen der Endschalter! *)
			T_ExchgParam.T_StationCommon.iZAxisFirstSetupStartButton_StepNr:=1;	(* Bitte StartTaste drücken für Prozedur zu starten! *)
			T_ExchgParam.T_StationCommon.iZAxisFirstSetup_ShowObjectNr:=1;
		END_IF;
	END_IF

	T_ExchgParam.T_StationCommon.rZAxisFirstSetup_OffsetSpinToDeskTop:=290.0;						(* 290mm muss eingerichtet werden und zwar distanz zwischen Spindel und Tischplatte *)
	rZAxisSetPosition:=T_ExchgParam.T_StationCommon.rZAxisFirstSetup_OffsetSpinToDeskTop - 190.0;	(* 190.0mm ist die Distanz zwischen Tischplatte und Spindel wo dann die Nullstellung definiert wird *)

	IF xTmpStationSetupAxisZFunction THEN
		CASE iStepHelpVisuFunction OF
		(* Erst Einrichtung der Z Axis *)
		1:	T_Visu.T_CtrleAction.xFunctionActive:=TRUE;
			T_CtrleBtStartStop.xForceSetStartButton:=TONWaitReadyStartButton.Q;
			IF xStartButton THEN
				TONWaitReadyStartButton(IN:=FALSE);
				T_ExchgParam.T_StationCommon.iZAxisFirstSetup_StepNr:=3;				(* Z Position wie unteres Bild setzen! *)
				T_ExchgParam.T_StationCommon.iZAxisFirstSetupStartButton_StepNr:=3;	(* Nachträglich Bitte StartTaste drücken um Position zu übernehmen *)
				T_ExchgParam.T_StationCommon.iZAxisFirstSetup_ShowObjectNr:=3;
				iStepHelpVisuFunction:=iStepHelpVisuFunction + 1;
				(* next step *)
				xTmpStepActionDone:=FALSE;
			END_IF;
		2:	T_CtrleBtStartStop.xForceSetStartButton:=TONWaitReadyStartButton.Q;
			IF xStartButton THEN
				TONWaitReadyStartButton(IN:=FALSE);
				T_ExchgParam.T_StationCommon.iZAxisFirstSetup_StepNr:=4;				(* Automatisches suchen des Z negativen Endschalter! *)
				T_ExchgParam.T_StationCommon.iZAxisFirstSetupStartButton_StepNr:=4;	(* Bitte StartTaste drücken um Bewegung auszulösen! *)
				T_ExchgParam.T_StationCommon.iZAxisFirstSetup_ShowObjectNr:=4;
				iStepHelpVisuFunction:=iStepHelpVisuFunction + 1;
			END_IF;
		(* Setzen der Nullposition der Z2 Achse *)
		3:	T_NovRam.T_Parameter.T_StationWork[gciStationSt1].T_AxisState.rPositionReferenceZAxis_Old:=	T_NovRam.T_Parameter.T_StationWork[gciStationSt1].T_AxisState.rPositionReferenceZAxis;
			IF NOT(T_NovRam.T_Parameter.T_StationWork[gciStationSt1].T_AxisState.xReferencedZAxis) THEN
				T_NovRam.T_Parameter.T_StationWork[gciStationSt1].T_AxisState.rPositionReferenceZAxis:=ptrActivStation^.THWWorkStation.TAxisZ.T_LiveValue.lrActualPosition + rZAxisSetPosition;
			ELSE
				T_NovRam.T_Parameter.T_StationWork[gciStationSt1].T_AxisState.rPositionReferenceZAxis:=	T_NovRam.T_Parameter.T_StationWork[gciStationSt1].T_AxisState.rPositionReferenceZAxis +
																																ptrActivStation^.THWWorkStation.TAxisZ.T_LiveValue.lrActualPosition +
																																rZAxisSetPosition;
			END_IF;
			T_NovRam.T_Parameter.T_StationWork[gciStationSt1].T_StProcess.rPositionEndMech:=0;
			ptrActivStation^.THWWorkStation.TAxisZ.T_CtrleSingle.iFunction:=11;	(* Position setzen *)
			ptrActivStation^.THWWorkStation.TAxisZ.T_CtrleSingle.rSetPosition:=(rZAxisSetPosition * -1.0);
			ptrActivStation^.THWWorkStation.TAxisZ.T_CtrleSingle.xExecute:=TRUE;
			iStepHelpVisuFunction:=iStepHelpVisuFunction + 1;
		4:	IF NOT(ptrActivStation^.THWWorkStation.TAxisZ.T_CtrleSingle.xExecute) AND ptrActivStation^.THWWorkStation.TAxisZ.T_CtrleSingle.xDone THEN
				T_NovRam.T_Parameter.T_StationWork[gciStationSt1].T_AxisState.xReferencedZAxis:=TRUE;
				iStepHelpVisuFunction:=iStepHelpVisuFunction + 1;
			END_IF;
		5:	xAction_SaveNovRAM:=TRUE;
			xBlockSetNovRamAction_End:=TRUE;
			iStepActionNovRam:=1;
			iStepHelpVisuFunction:=iStepHelpVisuFunction + 1;
		6:	IF NOT(xAction_SaveNovRAM) THEN
				xUpdateStationParameter:=TRUE;
				iStepHelpVisuFunction:=iStepHelpVisuFunction + 1;
			END_IF;
		7:	T_CtrleBtStartStop.xForceSetStartButton:=TONWaitReadyStartButton.Q;
			IF xStartButton THEN
				TONWaitReadyStartButton(IN:=FALSE);
				T_ExchgParam.T_StationCommon.iZAxisFirstSetup_StepNr:=4;				(* Automatisches suchen des Z negativen Endschalter! *)
				T_ExchgParam.T_StationCommon.iZAxisFirstSetupStartButton_StepNr:=5;	(* Ausmessung der Z Achse ist am durchführen... *)
				T_ExchgParam.T_StationCommon.iZAxisFirstSetup_ShowObjectNr:=4;
				iStepHelpVisuFunction:=iStepHelpVisuFunction + 1;
				ptrActivStation^.TControl.xExecute:=TRUE;
				ptrActivStation^.TControl.iFunctNr:=9;	(* Erstinitialisierung der Z Achse *)
				(* next step *)
				xTmpStepActionDone:=FALSE;
			END_IF;
		(* wait confirmation *)
		8:	IF NOT(xTmpStepActionDone) THEN
			(* release execution *)
				ptrActivStation^.TControl.xExecute:=FALSE;
				xTmpStepActionDone:=TRUE;
			ELSE
				IF ptrActivStation^.TControl.xDone THEN
					T_ExchgParam.T_StationCommon.iZAxisFirstSetup_StepNr:=5;				(* Nullstellung der Z Achse ist gesetzt! *)
					T_ExchgParam.T_StationCommon.iZAxisFirstSetupStartButton_StepNr:=6;	(* Bitte StartTaste drücken um Prozedur abzuschliessen! *)
					T_ExchgParam.T_StationCommon.iZAxisFirstSetup_ShowObjectNr:=5;
					(* action done *)
					iStepHelpVisuFunction:=iStepHelpVisuFunction + 1;
					xTmpStepActionDone:=FALSE;
				END_IF
			END_IF
		(* Anzeigen der Position für die Erstinitialisierung der Z Achse und dann Prozedur beenden *)
		9:	T_CtrleBtStartStop.xForceSetStartButton:=TONWaitReadyStartButton.Q;
			IF xStartButton THEN
				TONWaitReadyStartButton(IN:=FALSE);
				T_ExchgParam.T_StationCommon.iZAxisFirstSetup_StepNr:=1;				(* Setzen der Z Nullstellung und ausmessen der Endschalter! *)
				T_ExchgParam.T_StationCommon.iZAxisFirstSetupStartButton_StepNr:=1;	(* Bitte StartTaste drücken für Prozedur zu starten! *)
				T_ExchgParam.T_StationCommon.iZAxisFirstSetup_ShowObjectNr:=1;
				iStepHelpVisuFunction:=1;
				(* next step *)
				xTmpStepActionDone:=FALSE;
				xTmpStationSetupAxisZFunction:=FALSE;
				T_Visu.T_CtrleAction.xFunctionActive:=FALSE;
				T_StartUp.T_State.xBlockChangeMovementVisu:=FALSE;
				T_ExchgParam.T_Visu.T_Message.iState:=59;	(* Info: Funktion beendet ! *)
			END_IF;
		END_CASE;
	END_IF;

	IF (T_Visu.T_PlcParam.dwActualPage = gT_PageNumber.iWorkStation_Setup3) THEN
		T_ExchgParam.T_StationCommon.T_Param_StationWork.T_AxisState.rPositionNegLimitSwitchZAxis:=
												T_NovRam.T_Parameter.T_StationWork[gciStationSt1].T_AxisState.rPositionNegLimitSwitchZAxis;
		T_ExchgParam.T_StationCommon.T_Param_StationWork.T_AxisState.rPositionNegLimitSwitchZAxis_Old:=
												T_NovRam.T_Parameter.T_StationWork[gciStationSt1].T_AxisState.rPositionNegLimitSwitchZAxis_Old;
		T_ExchgParam.T_StationCommon.T_Param_StationWork.T_AxisState.rPositionReferenceZAxis:=
												T_NovRam.T_Parameter.T_StationWork[gciStationSt1].T_AxisState.rPositionReferenceZAxis;
		T_ExchgParam.T_StationCommon.T_Param_StationWork.T_AxisState.rPositionReferenceZAxis_Old:=
												T_NovRam.T_Parameter.T_StationWork[gciStationSt1].T_AxisState.rPositionReferenceZAxis_Old;
		T_ExchgParam.T_StationCommon.T_Param_StationWork.T_AxisState.xReferencedZAxis:=T_NovRam.T_Parameter.T_StationWork[gciStationSt1].T_AxisState.xReferencedZAxis;
		T_ExchgParam.T_StationCommon.xInitial_FirstSetupZ:=	T_NovRam.T_Parameter.T_StationWork[gciStationSt1].T_AxisState.xReferencedZAxis;
	END_IF;
END_ACTION
ACTION VisuFunction_Setup_Z_Axis_ToolGuide:
(* Ausführen von Stationsfunktionen für das Einrichten der Z Achse für das bestimmen der Z Achsen Position in Abhängigkeit der Position des oberen Führungsrohr *)
	IF xStationSetupAxisZFunctionToolGuide THEN
		(* Step  function station  *)
		CASE iStepAction OF
		(* Überprüfe zuerst ob die Stationen bereit stehen  *)
		1:	(* For start the procedure, it need the system level *)
			IF (T_ExchgParam.T_Visu.T_Level.iActLevel <> 2) THEN
				T_ExchgParam.T_Visu.T_Message.iState:=216;	(* Warnung: Diese Parameter können nur auf SystemLevel geändert werden ! *)
				iStepAction:=90;
				RETURN;
			END_IF;
			IF NOT(T_NovRam.T_Parameter.T_StationWork[gciStationSt1].T_AxisState.xReferencedZAxis) THEN
				T_ExchgParam.T_Visu.T_Message.iState:=294;	(* Warnung: Z Achse Ersteinrichtung zuerst durchführen ! *)
				iStepAction:=90;
				RETURN;
			END_IF;
			xTmp:=	ptrActivStation^.TControl.xDone
					AND ptrActivStation^.TControl.xRdy
					AND NOT(ptrActivStation^.TControl.xExecute)
					AND NOT(ptrActivStation^.TControl.xError)
					AND NOT(ptrActivStation^.TControl.xStop);
			(* next step *)
			IF xTmp THEN
				T_ExchgParam.T_StationCommon.iZAxisGuideTube_StepNr:=2;				(* Untere Anweisung durchführen! *)
				T_ExchgParam.T_StationCommon.iZAxisGuideTubeStartButton_StepNr:=2;		(* Nachträglich Bitte StartTaste drücken! *)
				T_ExchgParam.T_StationCommon.iZAxisGuideTube_ShowObjectNr:=2;
				iStepAction:=10;
				T_ExchgParam.T_Visu.T_Message.iState:=58;	(* Info: Funktion gestartet ! *)
			ELSE iStepAction:=95; END_IF
		(* Visu Ressource muss frei gegeben werden, da in dieser Prozedur noch zusätzliche VisuFunktionen benötigt werden *)
		10:	xTmpStationSetupAxisZFunctionToolGuide:=TRUE;
			iStepHelpVisuFunction:=1;
			T_StartUp.T_State.xBlockChangeMovementVisu:=TRUE;	(* Blockiere die Visu Navigation *)
			iStepAction:=90;
		(* action done *)
		90:	T_Visu.T_CtrleAction.xDone:=TRUE;
			T_Visu.T_CtrleAction.xNotReady:=FALSE;
			T_Visu.T_CtrleAction.xErr:=FALSE;
			T_Visu.T_CtrleAction.udiErrorID:=0;
			xStationSetupAxisZFunctionToolGuide:=FALSE;
		(* function not ready *)
		95:	TimerNotReady(IN:=TRUE);
			xStationSetupAxisZFunctionToolGuide:=FALSE;
		END_CASE
	ELSE
		IF NOT(xTmpStationSetupAxisZFunctionToolGuide) THEN
			T_ExchgParam.T_StationCommon.iZAxisGuideTube_StepNr:=1;				(* Setzen der abhängigkeit Z Achse und oberes Führungsrohr! *)
			T_ExchgParam.T_StationCommon.iZAxisGuideTubeStartButton_StepNr:=1;		(* Bitte StartTaste drücken für Prozedur zu starten! *)
			T_ExchgParam.T_StationCommon.iZAxisGuideTube_ShowObjectNr:=1;
		END_IF;
	END_IF

	T_NovRam.T_Parameter.T_StationWork[gciStationSt1].T_Z_TGuide.rDistanceTGuideToTableBoard:=250.0;	(* Distanz zwischen dem Schlitten des oberen Führungsrohr zur Tischplatte muss 250mm eingestellt werden *)
	T_NovRam.T_Parameter.T_StationWork[gciStationSt1].T_Z_TGuide.rScaleDefinedPos:=160.0;	(* Wenn der Schlitten des oberen Führungsrohr auf diese 250mm gesetzt ist, dann muss der Massstab so eingerichtet werden, dass es auf 160mm steht *)

	IF xTmpStationSetupAxisZFunctionToolGuide THEN
		CASE iStepHelpVisuFunction OF
		(* Erst Einrichtung der Z Axis *)
		1:	T_Visu.T_CtrleAction.xFunctionActive:=TRUE;
			T_CtrleBtStartStop.xForceSetStartButton:=TONWaitReadyStartButton.Q;
			IF xStartButton THEN
				TONWaitReadyStartButton(IN:=FALSE);
				T_ExchgParam.T_StationCommon.iZAxisGuideTube_StepNr:=3;				(* Untere Anweisung durchführen! *)
				T_ExchgParam.T_StationCommon.iZAxisGuideTubeStartButton_StepNr:=3;		(* Nachträglich Bitte StartTaste drücken! *)
				T_ExchgParam.T_StationCommon.iZAxisGuideTube_ShowObjectNr:=3;
				iStepHelpVisuFunction:=iStepHelpVisuFunction + 1;
				(* next step *)
				xTmpStepActionDone:=FALSE;
			END_IF;
		2:	T_CtrleBtStartStop.xForceSetStartButton:=TONWaitReadyStartButton.Q;
			IF xStartButton THEN
				TONWaitReadyStartButton(IN:=FALSE);
				T_ExchgParam.T_StationCommon.iZAxisGuideTube_StepNr:=4;				(* Untere Anweisung durchführen! *)
				T_ExchgParam.T_StationCommon.iZAxisGuideTubeStartButton_StepNr:=4;		(* Nachträglich Bitte StartTaste drücken! *)
				T_ExchgParam.T_StationCommon.iZAxisGuideTube_ShowObjectNr:=4;
				iStepHelpVisuFunction:=iStepHelpVisuFunction + 1;
			END_IF;
		3:	T_CtrleBtStartStop.xForceSetStartButton:=TONWaitReadyStartButton.Q;
			IF xStartButton THEN
				TONWaitReadyStartButton(IN:=FALSE);
				T_ExchgParam.T_StationCommon.iZAxisGuideTube_StepNr:=5;				(* Untere Anweisung durchführen! *)
				T_ExchgParam.T_StationCommon.iZAxisGuideTubeStartButton_StepNr:=5;		(* Nachträglich Bitte StartTaste drücken! *)
				T_ExchgParam.T_StationCommon.iZAxisGuideTube_ShowObjectNr:=5;
				iStepHelpVisuFunction:=iStepHelpVisuFunction + 1;
				T_NovRam.T_Parameter.T_StationWork[gciStationSt1].T_Z_TGuide.rToolLengthSetup:=
					T_ExchgParam.T_StationCommon.T_Param_StationWork.T_Z_TGuide.rToolLengthSetup;
			END_IF;
		4:	xAction_SaveNovRAM:=TRUE;
			xBlockSetNovRamAction_End:=TRUE;
			iStepActionNovRam:=1;
			iStepHelpVisuFunction:=iStepHelpVisuFunction + 1;
		5:	IF NOT(xAction_SaveNovRAM) THEN
				xUpdateStationParameter:=TRUE;
				iStepHelpVisuFunction:=iStepHelpVisuFunction + 1;
			END_IF;
		6:	T_CtrleBtStartStop.xForceSetStartButton:=TONWaitReadyStartButton.Q;
			IF xStartButton THEN
				TONWaitReadyStartButton(IN:=FALSE);
				T_ExchgParam.T_StationCommon.iZAxisGuideTube_StepNr:=6;				(* Untere Anweisung durchführen! *)
				T_ExchgParam.T_StationCommon.iZAxisGuideTubeStartButton_StepNr:=6;		(* Nachträglich Bitte StartTaste drücken! *)
				T_ExchgParam.T_StationCommon.iZAxisGuideTube_ShowObjectNr:=6;
				iStepHelpVisuFunction:=iStepHelpVisuFunction + 1;
				T_NovRam.T_Parameter.T_StationWork[gciStationSt1].T_Z_TGuide.rDistanceTGuideToTableBoardLess:=
					T_ExchgParam.T_StationCommon.T_Param_StationWork.T_Z_TGuide.rDistanceTGuideToTableBoardLess;
			END_IF;
		7:	xAction_SaveNovRAM:=TRUE;
			xBlockSetNovRamAction_End:=TRUE;
			iStepActionNovRam:=1;
			iStepHelpVisuFunction:=iStepHelpVisuFunction + 1;
		8:	IF NOT(xAction_SaveNovRAM) THEN
				xUpdateStationParameter:=TRUE;
				iStepHelpVisuFunction:=iStepHelpVisuFunction + 1;
			END_IF;
		9:	T_CtrleBtStartStop.xForceSetStartButton:=TONWaitReadyStartButton.Q;
			IF xStartButton THEN
				TONWaitReadyStartButton(IN:=FALSE);
				T_ExchgParam.T_StationCommon.iZAxisGuideTube_StepNr:=7;				(* Abhängigkeit ist gesetzt! *)
				T_ExchgParam.T_StationCommon.iZAxisGuideTubeStartButton_StepNr:=7;		(* Bitte StartTaste drücken um Prozedur abzuschliessen! *)
				T_ExchgParam.T_StationCommon.iZAxisGuideTube_ShowObjectNr:=7;
				iStepHelpVisuFunction:=iStepHelpVisuFunction + 1;
				T_NovRam.T_Parameter.T_StationWork[gciStationSt1].T_Z_TGuide.rOffset_Z_ToolGuide_Old:=
					T_NovRam.T_Parameter.T_StationWork[gciStationSt1].T_Z_TGuide.rOffset_Z_ToolGuide;
				T_NovRam.T_Parameter.T_StationWork[gciStationSt1].T_Z_TGuide.rOffset_Z_ToolGuide:=
					ptrTCommonAxis^.T_LiveValue.lrActualPosition;
			END_IF;
		10:	xAction_SaveNovRAM:=TRUE;
			xBlockSetNovRamAction_End:=TRUE;
			iStepActionNovRam:=1;
			iStepHelpVisuFunction:=iStepHelpVisuFunction + 1;
		11:	IF NOT(xAction_SaveNovRAM) THEN
				xUpdateStationParameter:=TRUE;
				iStepHelpVisuFunction:=iStepHelpVisuFunction + 1;
			END_IF;
		(* Anzeigen der Position für die Erstinitialisierung der Z Achse und dann Prozedur beenden *)
		12:	T_CtrleBtStartStop.xForceSetStartButton:=TONWaitReadyStartButton.Q;
			IF xStartButton THEN
				TONWaitReadyStartButton(IN:=FALSE);
				T_ExchgParam.T_StationCommon.iZAxisGuideTube_StepNr:=1;				(* Setzen der abhängigkeit Z Achse und oberes Führungsrohr! *)
				T_ExchgParam.T_StationCommon.iZAxisGuideTubeStartButton_StepNr:=1;		(* Bitte StartTaste drücken für Prozedur zu starten! *)
				T_ExchgParam.T_StationCommon.iZAxisGuideTube_ShowObjectNr:=1;
				iStepHelpVisuFunction:=1;
				(* next step *)
				xTmpStepActionDone:=FALSE;
				xTmpStationSetupAxisZFunctionToolGuide:=FALSE;
				T_Visu.T_CtrleAction.xFunctionActive:=FALSE;
				T_StartUp.T_State.xBlockChangeMovementVisu:=FALSE;
				T_ExchgParam.T_Visu.T_Message.iState:=59;	(* Info: Funktion beendet ! *)
			END_IF;
		END_CASE;
	END_IF;

	IF (T_Visu.T_PlcParam.dwActualPage = gT_PageNumber.iWorkStation_Setup3) THEN
		T_ExchgParam.T_StationCommon.T_Param_StationWork.T_Z_TGuide.rDistanceTGuideToTableBoard:=
												T_NovRam.T_Parameter.T_StationWork[gciStationSt1].T_Z_TGuide.rDistanceTGuideToTableBoard;
		T_ExchgParam.T_StationCommon.T_Param_StationWork.T_Z_TGuide.rOffset_Z_ToolGuide:=
												T_NovRam.T_Parameter.T_StationWork[gciStationSt1].T_Z_TGuide.rOffset_Z_ToolGuide;
		T_ExchgParam.T_StationCommon.T_Param_StationWork.T_Z_TGuide.rOffset_Z_ToolGuide_Old:=
												T_NovRam.T_Parameter.T_StationWork[gciStationSt1].T_Z_TGuide.rOffset_Z_ToolGuide_Old;
		T_ExchgParam.T_StationCommon.T_Param_StationWork.T_Z_TGuide.rScaleDefinedPos:=
												T_NovRam.T_Parameter.T_StationWork[gciStationSt1].T_Z_TGuide.rScaleDefinedPos;
		IF (T_ExchgParam.T_StationCommon.iZAxisGuideTube_ShowObjectNr <> 4) THEN
			T_ExchgParam.T_StationCommon.T_Param_StationWork.T_Z_TGuide.rToolLengthSetup:=
													T_NovRam.T_Parameter.T_StationWork[gciStationSt1].T_Z_TGuide.rToolLengthSetup;
		END_IF;
		IF (T_ExchgParam.T_StationCommon.iZAxisGuideTube_ShowObjectNr <> 5) THEN
			T_ExchgParam.T_StationCommon.T_Param_StationWork.T_Z_TGuide.rDistanceTGuideToTableBoardLess:=
													T_NovRam.T_Parameter.T_StationWork[gciStationSt1].T_Z_TGuide.rDistanceTGuideToTableBoardLess;
		END_IF;
	END_IF;
END_ACTION
ACTION VisuFunction_SetupPotentiometer:
(* Setup Potentiometer starten *)
	IF xSetupPotentiometer THEN
		CASE iStepAction OF
		(* check state *)
		1:	xTmp:=	TRUE;
			iStepPotentiometer:=0;
			(* next step *)
			IF xTmp THEN iStepAction:=10; ELSE iStepAction:=95; END_IF
		(* Set Value *)
		10:	(* For set the value, it need the system level *)
			IF (T_ExchgParam.T_Visu.T_Level.iActLevel <> 2) THEN
				T_ExchgParam.T_Visu.T_Message.iState:=216;	(* Warnung: Diese Parameter können nur auf SystemLevel geändert werden ! *)
				iStepAction:=90;
				RETURN;
			END_IF;
			CASE iStepPotentiometer OF
			0:	T_ExchgParam.T_Visu.T_Message.iState:=112;	(* Aufforderung: Position 0 am Poti einstellen und dann speichern *)
			1:	T_ExchgParam.T_Visu.T_Message.iState:=113;	(* Aufforderung: Position 1 am Poti einstellen und dann speichern *)
			2:	T_ExchgParam.T_Visu.T_Message.iState:=114;	(* Aufforderung: Position 2 am Poti einstellen und dann speichern *)
			3:	T_ExchgParam.T_Visu.T_Message.iState:=115;	(* Aufforderung: Position 3 am Poti einstellen und dann speichern *)
			4:	T_ExchgParam.T_Visu.T_Message.iState:=116;	(* Aufforderung: Position 4 am Poti einstellen und dann speichern *)
			5:	T_ExchgParam.T_Visu.T_Message.iState:=117;	(* Aufforderung: Position 5 am Poti einstellen und dann speichern *)
			6:	T_ExchgParam.T_Visu.T_Message.iState:=118;	(* Aufforderung: Position 6 am Poti einstellen und dann speichern *)
			7:	T_ExchgParam.T_Visu.T_Message.iState:=119;	(* Aufforderung: Position 7 am Poti einstellen und dann speichern *)
			8:	T_ExchgParam.T_Visu.T_Message.iState:=120;	(* Aufforderung: Position 8 am Poti einstellen und dann speichern *)
			9:	T_ExchgParam.T_Visu.T_Message.iState:=121;	(* Aufforderung: Position 9 am Poti einstellen und dann speichern *)
			10:	T_ExchgParam.T_Visu.T_Message.iState:=122;	(* Aufforderung: Position 10 am Poti einstellen und dann speichern *)
			END_CASE;
			iStepAction:=20;
		(* Display message to ask for confirmation *)
		20:	IF (T_ExchgParam.T_BtFunctionPanel.wActivBt = 32) THEN
				T_ExchgParam.T_Visu.T_Message.iState:=103;	(* Aufforderung: Speichern bestätigen <Enter>, abbrechen <Esc> ? *)
				iStepAction:=30;
			END_IF;
		(* waiting for key <Enter> or <Esc> *)
		30:	IF RisingEdgeKeyPanel_Enter.Q THEN
				iStepAction:=40;
				(* Display message *)
				T_ExchgParam.T_Visu.T_Message.iState:=3;	(* Info: Start speichern... *)
			ELSE
				IF RisingEdgeKeyPanel_Esc.Q THEN
					iStepAction:=90;
					T_ExchgParam.T_Visu.T_Message.iState:=202;	(* Warnung: Aktion abgebrochen ! *)
				END_IF
			END_IF
			(* An other message has been displayed *)
			IF (T_ExchgParam.T_Visu.T_Message.iState<>3) AND (T_ExchgParam.T_Visu.T_Message.iState<>103) AND (T_ExchgParam.T_Visu.T_Message.iState<>202) THEN iStepAction:=90; END_IF
		40:	T_NovRam.T_Parameter.T_Machine.adiPotentiometerValue[iStepPotentiometer]:=IiASpeedServoDrive;
			iStepAction:=50;
		50:	xAction_SaveNovRAM:=TRUE;
			xBlockSetNovRamAction_End:=TRUE;
			iStepActionNovRam:=1;
			iStepAction:=60;
		60:	IF NOT xAction_SaveNovRAM THEN
				T_ExchgParam.T_Visu.T_Message.iState:=25;	(* gewählte Pos ist nun gespeichert *)
				iStepPotentiometer:=iStepPotentiometer + 1;
				IF (iStepPotentiometer <= 10) THEN
					iStepAction:=10;
				ELSE
					iStepAction:=90;
					T_ExchgParam.T_Visu.T_Message.iState:=59;	(* Info: Funktion beendet ! *)
				END_IF;
			END_IF;
		(* action done *)
		90:	T_Visu.T_CtrleAction.xDone:=TRUE;
			T_Visu.T_CtrleAction.xNotReady:=FALSE;
			T_Visu.T_CtrleAction.xErr:=FALSE;
			T_Visu.T_CtrleAction.udiErrorID:=0;
			xSetupPotentiometer:=FALSE;
		(* cylinder not ready *)
		95:	TimerNotReady(IN:=TRUE);
			xSetupPotentiometer:=FALSE;
		END_CASE
	END_IF;

	FBLinearization_Potentiometer(	adi_X_MeasurePoint_Voltage:= T_NovRam.T_Parameter.T_Machine.adiPotentiometerValue,
								lr_X_Voltage:= IiASpeedServoDrive);

	T_ExchgParam.byOverride:=	REAL_TO_BYTE(FBLinearization_Potentiometer.lrScaledValuePercent);
	IF (T_ExchgParam.byOverride < 0) THEN
		T_ExchgParam.byOverride:=0;
	ELSIF (T_ExchgParam.byOverride > 100) THEN
		T_ExchgParam.byOverride:=100;
	END_IF;
	IF NOT(TProcess.T_Ctrle.xExecute) AND TProcess.T_Ctrle.xDone AND
	    NOT(TStation_Work_St1.TControl.xExecute) AND TStation_Work_St1.TControl.xDone AND
	    NOT(gxSetupFunctionActive) AND NOT(gxAxisAbsolutMovementActive) THEN
		T_ExchgParam.byOverride:=100;	(* Override nur wenn ein Prozess oder Station aktiv ist *)
	END_IF;
	TStation_Work_St1.THWWorkStation.TAxisZ.T_CtrleSingle.dwOverride:=T_ExchgParam.byOverride;

	(* Z Axis *)
	T_ExchgParam.T_TeachIn.arTeachSelStep[gciAxisZ_St1]:=	(1.0/100.0) * FBLinearization_Potentiometer.lrScaledValuePercent;
	IF (T_ExchgParam.T_TeachIn.arTeachSelStep[gciAxisZ_St1] < 0.01) THEN
		T_ExchgParam.T_TeachIn.arTeachSelStep[gciAxisZ_St1]:=0.01;
	END_IF;
	T_ExchgParam.T_TeachIn.arTeachSelVel[gciAxisZ_St1]:=	(20.0/100.0) * FBLinearization_Potentiometer.lrScaledValuePercent;
	IF (T_ExchgParam.T_TeachIn.arTeachSelVel[gciAxisZ_St1] < 0.1) THEN
		T_ExchgParam.T_TeachIn.arTeachSelVel[gciAxisZ_St1]:=0.1;
	END_IF;

	(* S Axis *)
	T_ExchgParam.T_TeachIn.arTeachSelStep[gciAxisS_St1]:=	(1.0/100.0) * FBLinearization_Potentiometer.lrScaledValuePercent;
	IF (T_ExchgParam.T_TeachIn.arTeachSelStep[gciAxisS_St1] < 0.01) THEN
		T_ExchgParam.T_TeachIn.arTeachSelStep[gciAxisS_St1]:=0.01;
	END_IF;
	T_ExchgParam.T_TeachIn.arTeachSelVel[gciAxisS_St1]:=	(20.0/100.0) * FBLinearization_Potentiometer.lrScaledValuePercent;
	IF (T_ExchgParam.T_TeachIn.arTeachSelVel[gciAxisS_St1] < 0.1) THEN
		T_ExchgParam.T_TeachIn.arTeachSelVel[gciAxisS_St1]:=0.1;
	END_IF;
END_ACTION
ACTION VisuFunction_SetupTorque:
(* Torque Offset -/+ *)
	IF xTorqueOffsetMinus OR xTorqueOffsetPlus THEN
		CASE iStepAction OF
		(* check state *)
		1:	xTmp:=	TRUE;
			(* next step *)
			IF xTmp THEN iStepAction:=10; ELSE iStepAction:=95; END_IF
		(* Set Value *)
		10:	IF xTorqueOffsetMinus THEN
				T_ExchgParam.T_AnalogSensTorque.rActual_Offset:=T_ExchgParam.T_AnalogSensTorque.rActual_Offset - 0.01;
			ELSE
				T_ExchgParam.T_AnalogSensTorque.rActual_Offset:=T_ExchgParam.T_AnalogSensTorque.rActual_Offset + 0.01;
			END_IF;
			iStepAction:=90;
		(* action done *)
		90:	T_Visu.T_CtrleAction.xDone:=TRUE;
			T_Visu.T_CtrleAction.xNotReady:=FALSE;
			T_Visu.T_CtrleAction.xErr:=FALSE;
			T_Visu.T_CtrleAction.udiErrorID:=0;
			xTorqueOffsetMinus:=xTorqueOffsetPlus:=FALSE;
		(* cylinder not ready *)
		95:	TimerNotReady(IN:=TRUE);
			xTorqueOffsetMinus:=xTorqueOffsetPlus:=FALSE;
		END_CASE
	END_IF;

(* Save Torque Scale *)
	IF xSaveTorqueScale THEN
		CASE iStepAction OF
		(* check state *)
		1:	xTmp:=	TRUE;
			(* next step *)
			IF xTmp THEN iStepAction:=10; ELSE iStepAction:=95; END_IF
		(* Set Value *)
		10:	(* For set the value, it need the system level *)
			IF (T_ExchgParam.T_Visu.T_Level.iActLevel <> 2) THEN
				T_ExchgParam.T_Visu.T_Message.iState:=216;	(* Warnung: Diese Parameter können nur auf SystemLevel geändert werden ! *)
				iStepAction:=90;
				RETURN;
			END_IF;
			iStepAction:=20;
		(* Display message to ask for confirmation *)
		20:	T_ExchgParam.T_Visu.T_Message.iState:=103;	(* Aufforderung: Speichern bestätigen <Enter>, abbrechen <Esc> ? *)
			iStepAction:=30;
		(* waiting for key <Enter> or <Esc> *)
		30:	IF RisingEdgeKeyPanel_Enter.Q THEN iStepAction:=40;
			ELSE
				IF RisingEdgeKeyPanel_Esc.Q THEN
					iStepAction:=90;
					T_ExchgParam.T_Visu.T_Message.iState:=202;	(* Warnung: Aktion abgebrochen ! *)
				END_IF
			END_IF
			(* An other message has been displayed *)
			IF (T_ExchgParam.T_Visu.T_Message.iState<>103) AND (T_ExchgParam.T_Visu.T_Message.iState<>202) THEN iStepAction:=90; END_IF
		40:	CASE T_ExchgParam.bToolSpindleActive OF
			1:	(* Maxon Spindel *)
				IF (T_ExchgParam.T_AnalogSensTorque.rMeasureDistance <> 0.0) THEN
					T_ExchgParam.T_AnalogSensTorque.rScaleFactor:=	IiAToolTorque_St1;
					T_NovRAM.T_Parameter.T_StationWork[gciStationSt1].T_TorqueSystem.rTorqueScaleFactor:=	T_ExchgParam.T_AnalogSensTorque.rScaleFactor;
				ELSE
					T_ExchgParam.T_AnalogSensTorque.rScaleFactor:=	0.0;
					T_NovRAM.T_Parameter.T_StationWork[gciStationSt1].T_TorqueSystem.rTorqueScaleFactor:=	T_ExchgParam.T_AnalogSensTorque.rScaleFactor;
				END_IF;
				T_NovRAM.T_Parameter.T_StationWork[gciStationSt1].T_TorqueSystem.rMeasureDistance:=T_ExchgParam.T_AnalogSensTorque.rMeasureDistance;
			END_CASE;
			iStepAction:=50;
		50:	xAction_SaveNovRAM:=TRUE;
			xBlockSetNovRamAction_End:=TRUE;
			iStepActionNovRam:=1;
			iStepAction:=60;
		60:	IF NOT xAction_SaveNovRAM THEN
				iStepAction:=90;
				T_ExchgParam.T_Visu.T_Message.iState:=59;	(* Info: Funktion beendet ! *)
			END_IF;
		(* action done *)
		90:	T_Visu.T_CtrleAction.xDone:=TRUE;
			T_Visu.T_CtrleAction.xNotReady:=FALSE;
			T_Visu.T_CtrleAction.xErr:=FALSE;
			T_Visu.T_CtrleAction.udiErrorID:=0;
			xSaveTorqueScale:=FALSE;
		(* cylinder not ready *)
		95:	TimerNotReady(IN:=TRUE);
			xSaveTorqueScale:=FALSE;
		END_CASE
	END_IF;

(* Save Torque Position *)
	IF xSaveTorquePosition THEN
		CASE iStepAction OF
		(* check state *)
		1:	xTmp:=	TRUE;
			(* next step *)
			IF xTmp THEN iStepAction:=10; ELSE iStepAction:=95; END_IF
		(* Set Value *)
		10:	iStepAction:=20;
		(* Display message to ask for confirmation *)
		20:	T_ExchgParam.T_Visu.T_Message.iState:=103;	(* Aufforderung: Speichern bestätigen <Enter>, abbrechen <Esc> ? *)
			iStepAction:=30;
		(* waiting for key <Enter> or <Esc> *)
		30:	IF RisingEdgeKeyPanel_Enter.Q THEN iStepAction:=40;
			ELSE
				IF RisingEdgeKeyPanel_Esc.Q THEN
					iStepAction:=90;
					T_ExchgParam.T_Visu.T_Message.iState:=202;	(* Warnung: Aktion abgebrochen ! *)
				END_IF
			END_IF
			(* An other message has been displayed *)
			IF (T_ExchgParam.T_Visu.T_Message.iState<>103) AND (T_ExchgParam.T_Visu.T_Message.iState<>202) THEN iStepAction:=90; END_IF
		40:	CASE T_ExchgParam.bToolSpindleActive OF
			1:	(* Maxon Spindel *)
				CASE T_ExchgParam.T_AnalogSensTorque.iSelectHC_Position OF
				0:	T_NovRAM.T_Parameter.T_StationWork[gciStationSt1].T_TorqueSystem.rTorquePosition_HC:=	T_ExchgParam.T_AnalogSensTorque.rActual_Position +
																							T_ExchgParam.T_AnalogSensTorque.rActual_Offset;
				1:	T_NovRAM.T_Parameter.T_StationWork[gciStationSt1].T_TorqueSystem.rTorquePosition_HCOverload:=	T_ExchgParam.T_AnalogSensTorque.rActual_Position +
																									T_ExchgParam.T_AnalogSensTorque.rActual_Offset;
				END_CASE;
			END_CASE;
			iStepAction:=50;
		50:	xAction_SaveNovRAM:=TRUE;
			xBlockSetNovRamAction_End:=TRUE;
			iStepActionNovRam:=1;
			iStepAction:=60;
		60:	IF NOT xAction_SaveNovRAM THEN
				iStepAction:=90;
				T_ExchgParam.T_Visu.T_Message.iState:=59;	(* Info: Funktion beendet ! *)
			END_IF;
		(* action done *)
		90:	T_Visu.T_CtrleAction.xDone:=TRUE;
			T_Visu.T_CtrleAction.xNotReady:=FALSE;
			T_Visu.T_CtrleAction.xErr:=FALSE;
			T_Visu.T_CtrleAction.udiErrorID:=0;
			xSaveTorquePosition:=FALSE;
		(* cylinder not ready *)
		95:	TimerNotReady(IN:=TRUE);
			xSaveTorquePosition:=FALSE;
		END_CASE
	END_IF;

	T_ExchgParam.T_AnalogSensTorque.rActual_Position:=	ptrTSensorTorque_St1^.T_CtrleCyl.T_Analog.rPosIn;
	IF (T_Visu.T_PlcParam.dwActualPage = gT_PageNumber.iWorkStation_Setup4) THEN
		CASE T_ExchgParam.bToolSpindleActive OF
		1:	(* Maxon Spindel *)
			CASE T_ExchgParam.T_AnalogSensTorque.iSelectHC_Position OF
			0:	T_ExchgParam.T_AnalogSensTorque.rSaved_Position:=T_NovRAM.T_Parameter.T_StationWork[gciStationSt1].T_TorqueSystem.rTorquePosition_HC;
			1:	T_ExchgParam.T_AnalogSensTorque.rSaved_Position:=T_NovRAM.T_Parameter.T_StationWork[gciStationSt1].T_TorqueSystem.rTorquePosition_HCOverload;
			END_CASE;
		END_CASE;
	ELSE
		T_ExchgParam.T_AnalogSensTorque.rActual_Offset:=0.0;
	END_IF;
END_ACTION
ACTION VisuFunction_SpecialFunction:
CASE T_ExchgParam.bToolSpindleActive OF
1:	(* Maxon Spindel *)
	IF (T_ExchgParam.T_StationCommon.bSelectCylinderConfig <= 1) THEN
			T_ExchgParam.T_StationCommon.bShowCylinderConfig:=1;	(* Ansicht Auslenkung SM Kopf *)
	ELSE
		IF T_ExchgParam.T_StationCommon.xToolSpindle_L_Connect THEN
			T_ExchgParam.T_StationCommon.bShowCylinderConfig:=4;	(* Ansicht Drehmoment L Kopf *)
		ELSE
			T_ExchgParam.T_StationCommon.bShowCylinderConfig:=3;	(* Ansicht Drehmoment SM Kopf *)
		END_IF;
	END_IF;
2:	(* Beckhoff Spindel L *)
	T_ExchgParam.T_StationCommon.bShowCylinderConfig:=2;	(* Ansicht Auslenkung L Kopf *)
3:	(* Beckhoff Spindel M *)
	T_ExchgParam.T_StationCommon.bShowCylinderConfig:=5;	(* Ansicht Auslenkung M Kopf *)
END_CASE;

IF xStationSetupAxisZFunctionToolGuide OR xTmpStationSetupAxisZFunctionToolGuide THEN
	T_ExchgParam.T_StationCommon.xBlockSelectZAxisProcedure:=TRUE;
	T_ExchgParam.T_StationCommon.iZAxisFirstSetup_ShowObjectNr:=0;
ELSIF xStationSetupAxisZFunction OR xTmpStationSetupAxisZFunction THEN
	T_ExchgParam.T_StationCommon.xBlockSelectZAxisProcedure:=TRUE;
	T_ExchgParam.T_StationCommon.iZAxisGuideTube_ShowObjectNr:=0;
ELSE
	T_ExchgParam.T_StationCommon.xBlockSelectZAxisProcedure:=FALSE;
	IF (T_ExchgParam.T_StationCommon.bSelectZAxisProcedure <= 1) THEN
		T_ExchgParam.T_StationCommon.iZAxisGuideTube_ShowObjectNr:=1;
		T_ExchgParam.T_StationCommon.iZAxisFirstSetup_ShowObjectNr:=0;
	ELSE
		T_ExchgParam.T_StationCommon.iZAxisGuideTube_ShowObjectNr:=0;
		T_ExchgParam.T_StationCommon.iZAxisFirstSetup_ShowObjectNr:=1;
	END_IF;
END_IF;

(* Auswahl Position Führungsrohr, Auswahl Abstand Führungsrohr, Auswahl Werkzeug oder Auswahl Führungsrohreinsatz *)
	IF xSelectConfigPosition_1 OR xSelectConfigPosition_2 OR xSelectConfigPosition_3 OR xSelectConfigPosition_4 THEN
		CASE iStepAction OF
		(* check state *)
		1:	xTmp:=	TRUE;
			(* next step *)
			IF xTmp THEN iStepAction:=10; ELSE iStepAction:=95; END_IF
		(* Set Value *)
		10:	IF xSelectConfigPosition_1 THEN
				T_ExchgParam.T_StationCommon.iSelectConfigPosition:=1;
			ELSIF xSelectConfigPosition_2 THEN
				T_ExchgParam.T_StationCommon.iSelectConfigPosition:=2;
			ELSIF xSelectConfigPosition_3 THEN
				T_ExchgParam.T_StationCommon.iSelectConfigPosition:=3;
			ELSE
				T_ExchgParam.T_StationCommon.iSelectConfigPosition:=4;
			END_IF;
			iStepAction:=90;
		(* action done *)
		90:	T_Visu.T_CtrleAction.xDone:=TRUE;
			T_Visu.T_CtrleAction.xNotReady:=FALSE;
			T_Visu.T_CtrleAction.xErr:=FALSE;
			T_Visu.T_CtrleAction.udiErrorID:=0;
			xSelectConfigPosition_1:=xSelectConfigPosition_2:=xSelectConfigPosition_3:=xSelectConfigPosition_4:=FALSE;
		(* cylinder not ready *)
		95:	TimerNotReady(IN:=TRUE);
			xSelectConfigPosition_1:=xSelectConfigPosition_2:=xSelectConfigPosition_3:=xSelectConfigPosition_4:=FALSE;
		END_CASE
	END_IF;

	IF (T_ExchgParam.T_StationCommon.iSelectConfigPosition <> iSelectConfigPosition) THEN
		iSelectConfigPosition:=T_ExchgParam.T_StationCommon.iSelectConfigPosition;
		xUpdateStationParameter:=TRUE;
	END_IF;

(* Speichern der Positionskonfiguration oder KonfigPos EIN/AUS *)
	IF xSaveConfigPosition OR xConfigPosOnOff THEN
		CASE iStepAction OF
		(* check state *)
		1:	xTmp:=	TRUE;
			(* next step *)
			IF xTmp THEN iStepAction:=10; ELSE iStepAction:=95; END_IF
		(* Display message to ask for confirmation *)
		10:	T_ExchgParam.T_Visu.T_Message.iState:=103;	(* Aufforderung: Speichern bestätigen <Enter>, abbrechen <Esc> ? *)
			iStepAction:=20;
		(* waiting for key <Enter> or <Esc> *)
		20:	IF RisingEdgeKeyPanel_Enter.Q THEN iStepAction:=30;
			ELSE
				IF RisingEdgeKeyPanel_Esc.Q THEN
					iStepAction:=90;
					T_ExchgParam.T_Visu.T_Message.iState:=202;	(* Warnung: Aktion abgebrochen ! *)
				END_IF
			END_IF
			(* An other message has been displayed *)
			IF (T_ExchgParam.T_Visu.T_Message.iState<>103) AND (T_ExchgParam.T_Visu.T_Message.iState<>202) THEN iStepAction:=90; END_IF
		30:	IF xSaveConfigPosition THEN
				IF (T_ExchgParam.T_StationCommon.iSelectConfigPosition = 1) THEN
					T_NovRam.T_Parameter.T_StationWork[1].T_StProcess.rPosToolGuid_Up:=T_ExchgParam.T_StationCommon.T_Param_StationWork.T_StProcess.rPosToolGuid_Up;
					T_NovRam.T_Parameter.T_StationWork[1].T_StProcess.rPosToolGuid_Down:=T_ExchgParam.T_StationCommon.T_Param_StationWork.T_StProcess.rPosToolGuid_Down;
				ELSIF (T_ExchgParam.T_StationCommon.iSelectConfigPosition = 2) THEN
					T_NovRam.T_Parameter.T_StationWork[1].T_StProcess.rDistanceToolGuide:=T_ExchgParam.T_StationCommon.T_Param_StationWork.T_StProcess.rDistanceToolGuide;
					T_NovRam.T_Parameter.T_StationWork[1].T_StProcess.rDistanceToolEndPos:=T_ExchgParam.T_StationCommon.T_Param_StationWork.T_StProcess.rDistanceToolEndPos;
				ELSIF (T_ExchgParam.T_StationCommon.iSelectConfigPosition = 3) THEN
					T_NovRam.T_Parameter.T_StationWork[1].T_StProcess.rLengthTool_Fixed:=T_ExchgParam.T_StationCommon.T_Param_StationWork.T_StProcess.rLengthTool_Fixed;
					T_NovRam.T_Parameter.T_StationWork[1].T_StProcess.rLengthTool_Work:=T_ExchgParam.T_StationCommon.T_Param_StationWork.T_StProcess.rLengthTool_Work;
				ELSIF (T_ExchgParam.T_StationCommon.iSelectConfigPosition = 4) THEN
					T_NovRam.T_Parameter.T_StationWork[1].T_StProcess.rLengthToolGuide:=T_ExchgParam.T_StationCommon.T_Param_StationWork.T_StProcess.rLengthToolGuide;
					T_NovRam.T_Parameter.T_StationWork[1].T_StProcess.rLengthAirTableBoard:=T_ExchgParam.T_StationCommon.T_Param_StationWork.T_StProcess.rLengthAirTableBoard;
				END_IF;
			ELSE
				T_NovRam.T_Parameter.T_StationWork[1].T_StProcess.xConfigActive:=NOT(T_NovRam.T_Parameter.T_StationWork[1].T_StProcess.xConfigActive);
			END_IF;
			iStepAction:=40;
		40:	xAction_SaveNovRAM:=TRUE;
			xBlockSetNovRamAction_End:=TRUE;
			iStepActionNovRam:=1;
			iStepAction:=50;
		50:	IF NOT xAction_SaveNovRAM THEN
				iStepAction:=90;
				T_ExchgParam.T_Visu.T_Message.iState:=59;	(* Info: Funktion beendet ! *)
			END_IF;
		(* action done *)
		90:	T_Visu.T_CtrleAction.xDone:=TRUE;
			T_Visu.T_CtrleAction.xNotReady:=FALSE;
			T_Visu.T_CtrleAction.xErr:=FALSE;
			T_Visu.T_CtrleAction.udiErrorID:=0;
			xSaveConfigPosition:=xConfigPosOnOff:=FALSE;
		(* cylinder not ready *)
		95:	TimerNotReady(IN:=TRUE);
			xSaveConfigPosition:=xConfigPosOnOff:=FALSE;
		END_CASE
	END_IF;

	gxProcessCylindricalAreaActive:=(T_NovRam.T_Parameter.T_StationWork[1].T_StProcess.rZPositionCylindricalArea <> 0.0);
	T_ExchgParam.T_StationCommon.xProcessCylindricalAreaActive:=gxProcessCylindricalAreaActive;
	IF NOT(gxProcessCylindricalAreaActive) THEN
		T_NovRam.T_Parameter.T_StationWork[1].T_StProcess.rZPositionCylindricalAreaStop:=0.0;
		T_ExchgParam.T_StationCommon.T_Param_StationWork.T_StProcess.rZPositionCylindricalAreaStop:=0.0;
	END_IF;

	T_ExchgParam.T_StationCommon.xSControllerActive:=(T_NovRam.T_Parameter.T_StationWork[1].T_StProcess.rWorkingSpindleSpeedMinMax <> 0.0);	(* Spindelregeler im Prozess Aktiv wenn dieser Wert nicht Null ist *)
	T_ExchgParam.T_StationCommon.xOControllerActive:=(T_NovRam.T_Parameter.T_StationWork[1].T_StProcess.rO_Ctrl_HystereseOffset <> 0.0);		(* Schnellhubregler im Prozess Aktiv wenn der Hysterese Offset nicht Null ist *)

	IF NOT(T_NovRam.T_Parameter.T_StationWork[1].T_StProcess.xConfigActive) THEN
		grZ_LoadPos:=T_NovRam.T_Parameter.T_StationWork[1].T_StProcess.rPositionLoad;
		grZ_WorkStartPos:=T_NovRam.T_Parameter.T_StationWork[1].T_StProcess.rPositionStartProc;
(*
		grZ_WorkEndPos:=T_NovRam.T_Parameter.T_StationWork[1].T_StProcess.rPositionEndProc;
*)
		IF NOT(gxProcessCylindricalAreaActive) THEN
			IF NOT(T_NovRam.T_Parameter.T_StationWork[1].T_StProcess.xPositionEndProcIncOnOff) THEN
				garPositionEndProcCalc[1]:=T_NovRam.T_Parameter.T_StationWork[1].T_StProcess.rPositionEndProc;
			ELSE
				IF (garPositionEndProcCalc[1] < T_NovRam.T_Parameter.T_StationWork[1].T_StProcess.rPositionEndProc) THEN
					garPositionEndProcCalc[1]:=T_NovRam.T_Parameter.T_StationWork[1].T_StProcess.rPositionEndProc;
				END_IF;
				IF (garPositionEndProcCalc[1] = 0.0) THEN
					garPositionEndProcCalc[1]:=T_NovRam.T_Parameter.T_StationWork[1].T_StProcess.rPositionEndProc;
				END_IF;
			END_IF;
			T_ExchgParam.T_StationCommon.rZPositionEndProc:=T_NovRam.T_Parameter.T_StationWork[1].T_StProcess.rPositionEndProc;
		ELSE
			(* Neuer Ablauf mit der Bestimmung des Zylindrischen Bereich ist aktiviert und deshalb gilt als End Position die Max Inkrement Position unabhängig ob mit oder ohne Inkrementierung *)
			IF NOT(T_NovRam.T_Parameter.T_StationWork[1].T_StProcess.xPositionEndProcIncOnOff) THEN
				garPositionEndProcCalc[1]:=T_NovRam.T_Parameter.T_StationWork[1].T_StProcess.rZPositionCylindricalArea;
			ELSE
				IF (garPositionEndProcCalc[1] < T_NovRam.T_Parameter.T_StationWork[1].T_StProcess.rZPositionCylindricalArea) THEN
					garPositionEndProcCalc[1]:=T_NovRam.T_Parameter.T_StationWork[1].T_StProcess.rZPositionCylindricalArea;
				END_IF;
				IF (garPositionEndProcCalc[1] = 0.0) THEN
					garPositionEndProcCalc[1]:=T_NovRam.T_Parameter.T_StationWork[1].T_StProcess.rZPositionCylindricalArea;
				END_IF;
			END_IF;
			T_ExchgParam.T_StationCommon.rZPositionEndProc:=T_NovRam.T_Parameter.T_StationWork[1].T_StProcess.rZPositionCylindricalArea;
		END_IF;
	ELSE
		grZ_LoadPos:=		T_NovRam.T_Parameter.T_StationWork[1].T_Z_TGuide.rOffset_Z_ToolGuide -
							(T_NovRam.T_Parameter.T_StationWork[1].T_StProcess.rLengthTool_Fixed - T_NovRam.T_Parameter.T_StationWork[1].T_Z_TGuide.rToolLengthSetup) -
							(T_NovRam.T_Parameter.T_StationWork[1].T_StProcess.rPosToolGuid_Up - T_NovRam.T_Parameter.T_StationWork[1].T_Z_TGuide.rScaleDefinedPos) +
							T_NovRam.T_Parameter.T_StationWork[1].T_StProcess.rLengthToolGuide -
							1.0;	(* Minus 1mm, damit das Wz nicht durch die ungenauigkeit aus dem Führungsrohr herausschaut *)
		grZ_WorkStartPos:=	T_NovRam.T_Parameter.T_StationWork[1].T_Z_TGuide.rOffset_Z_ToolGuide -
							(T_NovRam.T_Parameter.T_StationWork[1].T_StProcess.rLengthTool_Fixed - T_NovRam.T_Parameter.T_StationWork[1].T_Z_TGuide.rToolLengthSetup) +
							52.0 -
							T_NovRam.T_Parameter.T_StationWork[1].T_StProcess.rDistanceToolGuide -
							T_NovRam.T_Parameter.T_StationWork[1].T_StProcess.rLengthAirTableBoard +
							5.0;	(* Damit das Wz im unteren Führungsrohr ungefähr um 5mm drin ist *)
		grZ_WorkEndPos:=	T_NovRam.T_Parameter.T_StationWork[1].T_Z_TGuide.rOffset_Z_ToolGuide -
							(T_NovRam.T_Parameter.T_StationWork[1].T_StProcess.rLengthTool_Fixed - T_NovRam.T_Parameter.T_StationWork[1].T_Z_TGuide.rToolLengthSetup) +
							T_NovRam.T_Parameter.T_StationWork[1].T_Z_TGuide.rDistanceTGuideToTableBoardLess -
							T_NovRam.T_Parameter.T_StationWork[1].T_StProcess.rDistanceToolEndPos -
							T_NovRam.T_Parameter.T_StationWork[1].T_StProcess.rLengthAirTableBoard +
							T_NovRam.T_Parameter.T_StationWork[1].T_StProcess.rLengthTool_Work;
		IF NOT(T_NovRam.T_Parameter.T_StationWork[1].T_StProcess.xPositionEndProcIncOnOff) THEN
			garPositionEndProcCalc[1]:=grZ_WorkEndPos;
		ELSE
			IF (garPositionEndProcCalc[1] < grZ_WorkEndPos) THEN
				garPositionEndProcCalc[1]:=grZ_WorkEndPos;
			END_IF;
			IF (garPositionEndProcCalc[1] = 0.0) THEN
				garPositionEndProcCalc[1]:=grZ_WorkEndPos;
			END_IF;
		END_IF;
	END_IF;

	IF NOT(T_NovRam.T_Parameter.T_StationWork[1].T_StProcess.xCentringEndProcIncOnOff) THEN
		garCentringEndProcCalc[1]:=T_NovRam.T_Parameter.T_StationWork[1].T_StProcess.rCentringPosZ1Axis;
	ELSE
		IF (garCentringEndProcCalc[1] < T_NovRam.T_Parameter.T_StationWork[1].T_StProcess.rCentringPosZ1Axis) THEN
			garCentringEndProcCalc[1]:=T_NovRam.T_Parameter.T_StationWork[1].T_StProcess.rCentringPosZ1Axis;
		END_IF;
		IF (garCentringEndProcCalc[1] = 0.0) THEN
			garCentringEndProcCalc[1]:=T_NovRam.T_Parameter.T_StationWork[1].T_StProcess.rCentringPosZ1Axis;
		END_IF;
	END_IF;

	IF (T_Visu.T_PlcParam.dwActualPage <> gT_PageNumber.iAutoMode_ToolChange) AND (T_Visu.T_PlcParam.dwActualPage <> gT_PageNumber.iHandMode_Parameter) THEN
		T_ExchgParam.T_StationCommon.rPositionEndProcCalc:=	garPositionEndProcCalc[1];
		T_ExchgParam.T_StationCommon.rCentringEndProcCalc:=garCentringEndProcCalc[1];
	END_IF;

	IF T_NovRam.T_Parameter.T_StationWork[1].T_StProcess.xPositionEndProcIncOnOff THEN
		T_ExchgParam.T_StationCommon.xDisableChangeEndPos:=FALSE;
	ELSE
		T_ExchgParam.T_StationCommon.xDisableChangeEndPos:=TRUE;
	END_IF;

	IF T_NovRam.T_Parameter.T_StationWork[1].T_StProcess.xCentringEndProcIncOnOff THEN
		T_ExchgParam.T_StationCommon.xDisableCentringChangeEndPos:=FALSE;
	ELSE
		T_ExchgParam.T_StationCommon.xDisableCentringChangeEndPos:=TRUE;
	END_IF;

	xTmp:=	TProcess.T_Ctrle.xEnable AND
			NOT(TProcess.T_Ctrle.xExecute) AND
			(NOT(TProcess.T_Ctrle.xDone) OR
			TProcess.T_Ctrle.xError);
	T_ExchgParam.T_StationCommon.xDisableConfigPosition:=xTmp;




(* Regler Parameter speichern *)		(* IGS *)
IF xRegulatorOverlaySave THEN
	CASE iStepAction OF
	(* check state *)
	1:	(*iTmpSelectedStationAutomat:=giSelectedStationAutomat;*)
		xTmp:=	TRUE;
		(* next step *)
		IF xTmp THEN iStepAction:=20; ELSE iStepAction:=95; END_IF
	(* Display message to ask for confirmation *)
	20:	T_ExchgParam.T_Visu.T_Message.iState:=103;	(* Aufforderung: Speichern bestätigen <Enter>, abbrechen <Esc> ? *)
		iStepAction:=30;
	(* waiting for key <Enter> or <Esc> *)
	30:	IF RisingEdgeKeyPanel_Enter.Q THEN
			iStepAction:=40;
		ELSE
			IF RisingEdgeKeyPanel_Esc.Q THEN
				iStepAction:=90;
				T_ExchgParam.T_Visu.T_Message.iState:=202;	(* Warnung: Aktion abgebrochen ! *)
			END_IF
		END_IF
		(* An other message has been displayed *)
		IF ((T_ExchgParam.T_Visu.T_Message.iState<>103) AND (T_ExchgParam.T_Visu.T_Message.iState<>202)) (*OR (iTmpSelectedStationAutomat <> giSelectedStationAutomat)*) THEN iStepAction:=90; END_IF
	40:	IF (T_NovRAM.T_Parameter.T_StationWork[1].T_StProcess.iWorkControlType <= 1) THEN
			T_NovRAM.T_Parameter.T_StationWork[1].T_OnlineChange.rWorkingSpeedForward:=		T_ExchgParam.T_StationCommon.rSpeedZ_V1;
			T_NovRAM.T_Parameter.T_StationWork[1].T_OnlineChange.rTorqueLevelHC:=			T_ExchgParam.T_StationCommon.rTorqueZ_S4;
		ELSIF (T_NovRAM.T_Parameter.T_StationWork[1].T_StProcess.iWorkControlType = 2) THEN
			T_NovRAM.T_Parameter.T_StationWork[1].T_StProcess.rZ_PID_Torque:=T_ExchgParam.T_StationCommon.T_Param_StationWork.T_StProcess.rZ_PID_Torque;
			T_NovRAM.T_Parameter.T_StationWork[1].T_StProcess.rZ_PID_Kp:=T_ExchgParam.T_StationCommon.T_Param_StationWork.T_StProcess.rZ_PID_Kp;
			T_NovRAM.T_Parameter.T_StationWork[1].T_StProcess.rZ_PID_Ki:=T_ExchgParam.T_StationCommon.T_Param_StationWork.T_StProcess.rZ_PID_Ki;
			T_NovRAM.T_Parameter.T_StationWork[1].T_StProcess.rZ_PID_Kd:=T_ExchgParam.T_StationCommon.T_Param_StationWork.T_StProcess.rZ_PID_Kd;
			T_NovRAM.T_Parameter.T_StationWork[1].T_StProcess.rZ_PID_MinSpeed:=T_ExchgParam.T_StationCommon.T_Param_StationWork.T_StProcess.rZ_PID_MinSpeed;
			T_NovRAM.T_Parameter.T_StationWork[1].T_StProcess.rZ_PID_MaxSpeed:=T_ExchgParam.T_StationCommon.T_Param_StationWork.T_StProcess.rZ_PID_MaxSpeed;
			T_NovRAM.T_Parameter.T_StationWork[1].T_StProcess.iZ_PID_FilterM:=T_ExchgParam.T_StationCommon.T_Param_StationWork.T_StProcess.iZ_PID_FilterM;
		ELSE
			T_NovRAM.T_Parameter.T_StationWork[1].T_OnlineChange.rWorkingSpeedForward:=		T_ExchgParam.T_StationCommon.rSpeedZ_V1;
			T_NovRAM.T_Parameter.T_StationWork[1].T_OnlineChange.rTorqueLevelHC:=			T_ExchgParam.T_StationCommon.rTorqueZ_S4;
			T_NovRAM.T_Parameter.T_StationWork[1].T_StProcess.rZ_D_Kd:=T_ExchgParam.T_StationCommon.T_Param_StationWork.T_StProcess.rZ_D_Kd;
			T_NovRAM.T_Parameter.T_StationWork[1].T_StProcess.iZ_D_FilterM:=T_ExchgParam.T_StationCommon.T_Param_StationWork.T_StProcess.iZ_D_FilterM;
		END_IF;
		iStepAction:=50;
	50:	xAction_SaveNovRAM:=TRUE;
		xBlockSetNovRamAction_End:=TRUE;
		iStepActionNovRam:=1;
		iStepAction:=60;
	60:	IF NOT xAction_SaveNovRAM THEN
			iStepAction:=90;
			T_ExchgParam.T_Visu.T_Message.iState:=59;	(* Info: Funktion beendet ! *)
		END_IF;
	(* action done *)
	90:	T_Visu.T_CtrleAction.xDone:=TRUE;
		T_Visu.T_CtrleAction.xNotReady:=FALSE;
		T_Visu.T_CtrleAction.xErr:=FALSE;
		T_Visu.T_CtrleAction.udiErrorID:=0;
		xRegulatorOverlaySave:=FALSE;
		(*IF (iTmpSelectedStationAutomat <> giSelectedStationAutomat) THEN
			T_ExchgParam.T_Visu.T_Message.iState:=202;	(* Aktion abgebrochen *)
		END_IF;*)
	(* cylinder not ready *)
	95:	TimerNotReady(IN:=TRUE);
		xRegulatorOverlaySave:=FALSE;
	END_CASE
END_IF;

(* Auswahl Konventioneller Regler, Adaptive Voschub Regler oder Konventioneller PD Regler *)
IF xRegulatorType1 OR xRegulatorType2 OR xRegulatorType3 THEN
	CASE iStepAction OF
	(* check state *)
	1:	(*iTmpSelectedStationAutomat:=giSelectedStationAutomat;*)
		xTmp:=	TRUE;
		(* next step *)
		IF xTmp THEN iStepAction:=20; ELSE iStepAction:=95; END_IF
	(* Display message to ask for confirmation *)
	20:	T_ExchgParam.T_Visu.T_Message.iState:=103;	(* Aufforderung: Speichern bestätigen <Enter>, abbrechen <Esc> ? *)
		iStepAction:=30;
	(* waiting for key <Enter> or <Esc> *)
	30:	IF RisingEdgeKeyPanel_Enter.Q THEN
			iStepAction:=40;
		ELSE
			IF RisingEdgeKeyPanel_Esc.Q THEN
				iStepAction:=90;
				T_ExchgParam.T_Visu.T_Message.iState:=202;	(* Warnung: Aktion abgebrochen ! *)
			END_IF
		END_IF
		(* An other message has been displayed *)
		IF ((T_ExchgParam.T_Visu.T_Message.iState<>103) AND (T_ExchgParam.T_Visu.T_Message.iState<>202)) (*OR (iTmpSelectedStationAutomat <> giSelectedStationAutomat)*) THEN iStepAction:=90; END_IF
	40:	IF xRegulatorType1 THEN
			T_NovRAM.T_Parameter.T_StationWork[1].T_StProcess.iWorkControlType:=1;
		ELSIF xRegulatorType2 THEN
			T_NovRAM.T_Parameter.T_StationWork[1].T_StProcess.iWorkControlType:=2;
		ELSE
			T_NovRAM.T_Parameter.T_StationWork[1].T_StProcess.iWorkControlType:=3;
		END_IF;
		T_ExchgParam.T_StationCommon.T_Param_StationWork.T_StProcess.iWorkControlType:=T_NovRAM.T_Parameter.T_StationWork[1].T_StProcess.iWorkControlType;
		iStepAction:=50;
	50:	xAction_SaveNovRAM:=TRUE;
		xBlockSetNovRamAction_End:=TRUE;
		iStepActionNovRam:=1;
		iStepAction:=60;
	60:	IF NOT xAction_SaveNovRAM THEN
			iStepAction:=90;
			T_ExchgParam.T_Visu.T_Message.iState:=59;	(* Info: Funktion beendet ! *)
		END_IF;
	(* action done *)
	90:	T_Visu.T_CtrleAction.xDone:=TRUE;
		T_Visu.T_CtrleAction.xNotReady:=FALSE;
		T_Visu.T_CtrleAction.xErr:=FALSE;
		T_Visu.T_CtrleAction.udiErrorID:=0;
		xRegulatorType1:=xRegulatorType2:=xRegulatorType3:=FALSE;
	(* cylinder not ready *)
	95:	TimerNotReady(IN:=TRUE);
		xRegulatorType1:=xRegulatorType2:=xRegulatorType3:=FALSE;
	END_CASE
END_IF;

T_ExchgParam.T_StationCommon.rController2_MinSpeed:=	T_Profile.T_Profile_MinMax.T_Max.rWorkingSpeedForward * -1.0;

IF (T_Visu.T_PlcParam.dwActualPage <> gT_PageNumber.iHandMode_RegulatorPara) (*OR RisingEdgeStationNr.Q*) THEN
	T_ExchgParam.T_StationCommon.rSpeedZ_V1:=TStation_Work_St1.THWWorkStation.TCtrlWork.rSpeedZ_V1;
	T_ExchgParam.T_StationCommon.rSpeedZ_V3:=TStation_Work_St1.THWWorkStation.TCtrlWork.rSpeedZ_V3;
	T_ExchgParam.T_StationCommon.rTorqueZ_S1:=TStation_Work_St1.THWWorkStation.TCtrlWork.rTorqueZ_S1;
	T_ExchgParam.T_StationCommon.rTorqueZ_S4:=TStation_Work_St1.THWWorkStation.TCtrlWork.rTorqueZ_S4;
	T_ExchgParam.T_StationCommon.iProgressBar_Torque:=TStation_Work_St1.THWWorkStation.TCtrlWork.iProgressBar_Torque;
	T_ExchgParam.T_StationCommon.iProgressBar_ZPos:=TStation_Work_St1.THWWorkStation.TCtrlWork.iProgressBar_ZPos;
	T_ExchgParam.T_StationCommon.iProgressBar_ZVel:=TStation_Work_St1.THWWorkStation.TCtrlWork.iProgressBar_ZVel;
	T_ExchgParam.T_StationCommon.xTorqueAfterHC_Min_Overlimit:=TStation_Work_St1.THWWorkStation.TCtrlWork.xTorqueAfterHC_Min_Overlimit;
	T_ExchgParam.T_StationCommon.xTorqueAfterHC_Max_Overlimit:=TStation_Work_St1.THWWorkStation.TCtrlWork.xTorqueAfterHC_Max_Overlimit;
END_IF;
END_ACTION
ACTION VisuFunction_SpindleBurnIn:
(* Ausführen der Stationsfunktion für den BurnIn der Spindeln über ausgewählte Stationen *)
	IF xStationSpindleBurnInFunction THEN
		TONElapsedBurnInTime(IN:=TRUE,PT:=T#99999s);
		T_ExchgParam.T_SpindleBurnIn.tTimeElapsed:=TONElapsedBurnInTime.ET;
		(* Step  function station  *)
		CASE iStepAction OF
		(* Überprüfe zuerst ob die ausgewählten Stationen bereit stehen  *)
		1:	xTmp:=	(ptrActivStation^.TControl.xDone
					AND ptrActivStation^.TControl.xRdy
					AND NOT(ptrActivStation^.TControl.xExecute)
					AND NOT(ptrActivStation^.TControl.xError)
					AND NOT(ptrActivStation^.TControl.xStop)
					AND T_ExchgParam.T_SafetyCtrl.xSetupOperateB_EnergyON);
			(* next step *)
			IF xTmp THEN iStepAction:=10; ELSE iStepAction:=95; END_IF
		(* determin function number *)
		10:	ptrActivStation^.TControl.iFunctNr:=8;	(* Spindle Burn-In *)
			ptrActivStation^.TControl.xExecute:=TRUE;
			(* next step *)
			iStepAction:=20;
			(* next step *)
			xStepActionDone:=FALSE;
			T_ExchgParam.T_Visu.T_Message.iState:=63;	(* Info: BurnIn Funktion gestartet ! *)
		(* wait confirmation *)
		20:	IF NOT(xStepActionDone) THEN
			(* release execution *)
				ptrActivStation^.TControl.xExecute:=FALSE;
				xStepActionDone:=TRUE;
			ELSE
				xTmp:=	NOT(ptrActivStation^.TControl.xExecute) AND ptrActivStation^.TControl.xDone;
				IF xTmp THEN
					(* action done *)
					iStepAction:=90;
					xStepActionDone:=FALSE;
					T_ExchgParam.T_Visu.T_Message.iState:=64;	(* Info: BurnIn Funktion beendet ! *)
				END_IF
			END_IF
		(* action done *)
		90:	T_Visu.T_CtrleAction.xDone:=TRUE;
			T_Visu.T_CtrleAction.xNotReady:=FALSE;
			T_Visu.T_CtrleAction.xErr:=FALSE;
			T_Visu.T_CtrleAction.udiErrorID:=0;
			xStationSpindleBurnInFunction:=FALSE;
		(* function not ready *)
		95:	TimerNotReady(IN:=TRUE);
			xStationSpindleBurnInFunction:=FALSE;
		END_CASE
	ELSE
		TONElapsedBurnInTime(IN:=FALSE);
	END_IF
END_ACTION
ACTION VisuFunction_StationFunction:
(* Ausführen von Stationsfunktionen der Bearbeitungsstation oder des Handling *)
	IF xStationWorkFunction THEN
		(* Step  function station  *)
		CASE iStepAction OF
		1:	ptrActivStation_Function1:=ADR(TStation_Work_St1);
			IF NOT(T_NovRam.T_Parameter.T_StationWork[gciStationSt1].T_AxisState.xReferencedZAxis) THEN
				T_ExchgParam.T_Visu.T_Message.iState:=294;	(* Warnung: Z Achse Ersteinrichtung zuerst durchführen ! *)
				iStepAction:=90;
			ELSE
				FBGetStationFunctionNr(	iVisuFunctionNr:= T_ExchgParam.T_FunctionCommon.iFunctionNrMicrohead);
				iStationFunctionNr:=FBGetStationFunctionNr.iWorkStation_FunctionNr;
				iStepAction:=10;
				T_Visu.T_CtrleAction.xFunctionActive:=TRUE;
				ptrActivStation_Function1:=ADR(TStation_Work_St1);
			END_IF;
		(* check station state *)
		10:	xTmp:=	ptrActivStation_Function1^.TControl.xDone
					AND ptrActivStation_Function1^.TControl.xRdy
					AND NOT(ptrActivStation_Function1^.TControl.xExecute)
					AND NOT(ptrActivStation_Function1^.TControl.xError)
					AND NOT(ptrActivStation_Function1^.TControl.xStop);
			(* next step *)
			IF xTmp THEN
				iStepAction:=11;
			ELSE iStepAction:=95; END_IF
		(* determin function number *)
		11:	ptrActivStation_Function1^.TControl.iFunctNr:=iStationFunctionNr;
			T_ExchgParam.T_Visu.T_Message.iState:=58;	(* Info: Funktion gestartet ! *)
			(* Auffangen der Funktion ToolRotation *)
			ptrActivStation_Function1^.TControl.xExecute:=TRUE;
			iStepAction:=12;
			(* next step *)
			xStepActionDone:=FALSE;
		(* wait confirmation *)
		12:	IF NOT(xStepActionDone) THEN
			(* release execution *)
				ptrActivStation_Function1^.TControl.xExecute:=FALSE;
				xStepActionDone:=TRUE;
			ELSE
				IF ptrActivStation_Function1^.TControl.xDone THEN
					(* action done *)
					iStepAction:=90;
					xStepActionDone:=FALSE;
					T_ExchgParam.T_Visu.T_Message.iState:=59;	(* Info: Funktion beendet ! *)
				END_IF
			END_IF
		(* action done *)
		90:	T_Visu.T_CtrleAction.xDone:=TRUE;
			T_Visu.T_CtrleAction.xNotReady:=FALSE;
			T_Visu.T_CtrleAction.xErr:=FALSE;
			T_Visu.T_CtrleAction.udiErrorID:=0;
			xStationWorkFunction:=FALSE;
			T_Visu.T_CtrleAction.xFunctionActive:=FALSE;
		(* function not ready *)
		95:	TimerNotReady(IN:=TRUE);
			xStationWorkFunction:=FALSE;
			T_Visu.T_CtrleAction.xFunctionActive:=FALSE;
		END_CASE
	END_IF
END_ACTION
ACTION VisuFunction_StationStop:
(* Stoppen von Stationsfunktionen von rechter und linker Arbeitsstation *)
	IF xStationStop THEN
		(* Step  function station stop  *)
		CASE iStepAction OF
		(* Überprüfe zuerst welche Stationen gestoppt werden müssen  *)
		1:	iCheckStationNr:=1;
			ptrActivStation_FunctionStop:=ADR(TStation_Work_St1);
			iStepAction:=10;
		10:	IF (iCheckStationNr = 1) THEN ptrActivStation_FunctionStop:=ADR(TStation_Work_St1);
			ELSE
				iStepAction:=30;
				iCheckStationNr:=1;
				iStationNrReady:=0;
				RETURN;
			END_IF;
			xTmp:=	NOT(ptrActivStation_FunctionStop^.TControl.xDone)
					AND ptrActivStation_FunctionStop^.TControl.xRdy
					AND NOT(ptrActivStation_FunctionStop^.TControl.xExecute)
					AND NOT(ptrActivStation_FunctionStop^.TControl.xError)
					AND NOT(ptrActivStation_FunctionStop^.TControl.xStop);
			IF xTmp THEN
				(* Mindestens eine Station kann gestoppt werden *)
				iStepAction:=20;
			ELSE
				iCheckStationNr:=iCheckStationNr + 1;
			END_IF
		20:	ptrActivStation_FunctionStop^.TControl.xStop:=TRUE;
			iCheckStationNr:=iCheckStationNr + 1;
			(* next step *)
			iStepAction:=10;
		30:	IF (iCheckStationNr = 1) THEN ptrActivStation_FunctionStop:=ADR(TStation_Work_St1);END_IF;
			xTmp:=	(ptrActivStation_FunctionStop^.TControl.xDone OR ptrActivStation_FunctionStop^.TControl.xError)
					AND ptrActivStation_FunctionStop^.TControl.xRdy
					AND NOT(ptrActivStation_FunctionStop^.TControl.xExecute);
			IF xTmp THEN
				iStationNrReady:=iStationNrReady + 1;
			END_IF;
			iCheckStationNr:=iCheckStationNr + 1;
			IF (iCheckStationNr > 14) THEN
				IF (iStationNrReady = 14) THEN
					(* Alle Stationen sind gestoppt *)
					(* next step *)
					iStepAction:=40;
				ELSE
					(* Mindestens eine Station ist noch nicht gestoppt *)
					iCheckStationNr:=1;
					iStationNrReady:=0;
				END_IF;
			END_IF;
		(* Alle Stationen sind gestoppt. Nun müssen noch alle Achsen überprüft werden ob sie gestoppt sind *)
		40:	IF NOT(ptrTAxisZ_St1^.T_CtrleSingle.xNotMoving) AND NOT(ptrTAxisZ_St1^.T_CtrleSingle.xErr) THEN
				ptrTAxisZ_St1^.T_CtrleSingle.iFunction:=5;
				ptrTAxisZ_St1^.T_CtrleSingle.xExecute:=TRUE;
			END_IF;
			IF NOT(ptrTAxisS_St1^.T_CtrleSingle.xNotMoving) AND NOT(ptrTAxisS_St1^.T_CtrleSingle.xErr) THEN
				ptrTAxisS_St1^.T_CtrleSingle.iFunction:=5;
				ptrTAxisS_St1^.T_CtrleSingle.xExecute:=TRUE;
			END_IF;
			iStepAction:=50;
		(* Warte bis alle Achsen stehen *)
		50:	xTmp:=	(NOT(ptrTAxisZ_St1^.T_CtrleSingle.xExecute) AND (ptrTAxisZ_St1^.T_CtrleSingle.xDone OR ptrTAxisZ_St1^.T_CtrleSingle.xErr)) AND
					(NOT(ptrTAxisS_St1^.T_CtrleSingle.xExecute) AND (ptrTAxisS_St1^.T_CtrleSingle.xDone OR ptrTAxisS_St1^.T_CtrleSingle.xErr));
			IF xTmp THEN
				(* action done *)
				iStepAction:=90;
				T_ExchgParam.T_Visu.T_Message.iState:=274;	(* Warnung: Funktion wurde gestoppt ! *)
			END_IF;
		(* action done *)
		90:	T_Visu.T_CtrleAction.xFunctionActive:=FALSE;
			T_StartUp.T_State.xBlockChangeMovementVisu:=FALSE;
			T_Visu.T_CtrleAction.xDone:=TRUE;
			T_Visu.T_CtrleAction.xNotReady:=FALSE;
			T_Visu.T_CtrleAction.xErr:=FALSE;
			T_Visu.T_CtrleAction.udiErrorID:=0;
			xStationStop:=FALSE;
		(* function not ready *)
		95:	T_StartUp.T_State.xBlockChangeMovementVisu:=FALSE;
			TimerNotReady(IN:=TRUE);
			xStationStop:=FALSE;

		END_CASE;
	END_IF;

